PROGRAM Programa
VAR
    ToffPulse_1s : TON;
    TonPulse_1s : TON;
    ToffPulse_100ms : TON;
    TonPulse_100ms : TON;
    ToffPulse_2s : TON;
    TonPulse_2s : TON;
    ToffPulse_5s : TON;
    TonPulse_5s : TON;
    ToffPulse_10ms : TON;
    TonPulse_10ms : TON;
    ToffPulse_30s : TON;
    TonPulse_30s : TON;
    DelayRobotStep1 : TON;
    DelayRobotStep2 : TON;
    DelayRobotStep3 : TON;
    DelayRobotStep4 : TON;
    DelayRobotStep5 : TON;
    DelayRobotStep6 : TON;
    DelayRobotStep7 : TON;
    DelayRobotStep8 : TON;
    Motor110M1 : CmdLenzeI550;
    TimeResetAlarme : TON;
    Motor111M1 : CmdLenzeI550;
    Motor120M1 : CmdLenzeI550;
    Motor211M1 : CmdLenzeI550;
    Motor212M1 : CmdLenzeI550;
    Motor213M1 : CmdLenzeI550;
    Motor221M1 : CmdLenzeI550;
    Motor222M1 : CmdLenzeI550;
    Motor223M1 : CmdLenzeI550;
    Motor230M1 : CmdLenzeI550;
    Motor240M1 : CmdLenzeI550;
    Motor250M1 : CmdLenzeI550;
    Valve110V : CmdValve;
    Delay110M1Full : TON;
    Delay110VStep1 : TON;
    ncteste : BOOL;
    DelayAE110V : TON;
    Valve111V : CmdValve;
    DelayAE111V : TON;
    Delay111VStep4 : TON;
    DelayAE121V : TON;
    Valve121V : CmdValve;
    Delay121VStep4 : TON;
    DelayAE122V : TON;
    Delay122VStep4 : TON;
    DelayAE123V : TON;
    Valve122V : CmdValve;
    Delay123VStep4 : TON;
    DelayAE211V : TON;
    Valve211V : CmdValve;
    Delay211VStep1 : TON;
    DelayAE212V : TON;
    Valve212V : CmdValve;
    Delay212VStep1 : TON;
    DelayAE213V : TON;
    Valve213V : CmdValve;
    Delay213VStep1 : TON;
    Delay211M1Full : TON;
    Delay212M1Full : TON;
    Delay213M1Full : TON;
    Delay221M1Step2 : TON;
    Alarme_G_221M1 : CheckAlarmeEquip;
    Delay221M1Step4 : TimerPulse;
    Delay221M1Step9 : TON;
    Delay221M1Step11 : TimerPulse;
    Delay221M1Step16 : TimerPulse;
    Delay211M1Empty : TON;
    Delay212M1Empty : TON;
    Delay213M1Empty : TON;
    Delay211M1TimeOut : TON;
    Delay212M1TimeOut : TON;
    Delay213M1TimeOut : TON;
    Delay110M1TimeOut : TON;
    Alarme_G_230M1 : CheckAlarmeEquip;
    Delay230M1Step4 : TimerPulse;
    Delay230M1Step2 : TON;
    Delay221M1Step18 : TON;
    Delay230M1Step13 : TON;
    Delay230M1Step16 : TON;
    Delay221M1Step19 : TON;
    Alarme_G_222M1 : CheckAlarmeEquip;
    Delay222M1Step19 : TON;
    Delay222M1Step18 : TON;
    Delay222M1Step16 : TimerPulse;
    Delay222M1Step11 : TimerPulse;
    Delay222M1Step9 : TON;
    Delay222M1Step4 : TimerPulse;
    Delay222M1Step2 : TON;
    Alarme_G_223M1 : CheckAlarmeEquip;
    Delay223M1Step19 : TON;
    Delay223M1Step18 : TON;
    Delay223M1Step16 : TimerPulse;
    Delay223M1Step11 : TimerPulse;
    Delay223M1Step9 : TON;
    Delay223M1Step4 : TimerPulse;
    Delay223M1Step2 : TON;
    Delay111M1Step2 : TON;
    Delay111M1Step3 : TimerPulse;
    Delay111M1Step10 : TimerPulse;
    Delay111M1Step11 : TimerPulse;
    Delay111M1Step12 : TON;
    Delay111M1Step13 : TON;
    Delay111M1Step19 : TON;
    Delay111M1Step20 : TON;
    Read111U1 : EAN13Read;
    TimeOut111M1Step15 : TON;
    Delay111M1Step14 : TON;
    Delay120M1Step2 : TON;
    Delay120M1Step3 : TimerPulse;
    Delay120M1Step4 : TON;
    Delay120M1Step9 : TON;
    Delay120M1Step19 : TON;
    Delay111M1Step21 : TON;
    Delay120M1Step10 : TimerPulse;
    Delay120M1Step11 : TimerPulse;
    Delay120M1Step13 : TimerPulse;
    Delay120M1Step14 : TimerPulse;
    Delay120M1Step17 : TimerPulse;
    Delay120M1Step16 : TimerPulse;
    Alarme_G_240M1 : CheckAlarmeEquip;
    Delay240M1Step2 : TON;
    Delay240M1Step4 : TimerPulse;
    Delay240M1Step5 : TON;
    Delay240M1Step8 : TON;
    Delay240M1Step12 : TON;
    Alarme_G_250M1 : CheckAlarmeEquip;
    Delay250M1Step5 : TON;
    Delay250M1Step4 : TimerPulse;
    Delay250M1Step2 : TON;
    Delay250M1Step21 : TON;
    Delay250M1Step20 : TON;
    Delay250M1Step19 : TON;
    TimeOut250M1Step15 : TON;
    Delay250M1Step14 : TON;
    Delay250M1Step13 : TON;
    Delay250M1Step12 : TON;
    Delay250M1Step11 : TimerPulse;
    Delay250M1Step10 : TimerPulse;
    DelayAE251V : TON;
    Valve251V : CmdValve;
    Delay251VStep4 : TON;
    DelayAE252V : TON;
    Valve252V : CmdValve;
    Delay252VStep4 : TON;
    Delay250M1Step23 : TON;
    TimeMax251VStep3 : TON;
    TimeMax252VStep3 : TON;
    Delay250M1Step28 : TON;
    RstEthercat : ResetECError;
    RstPLC : ResetPLCError;
    CmdICM_540 : CmdICM;
    Motor540M1 : CmdMotor;
    Motor540M2 : CmdMotor;
    Motor610M1 : CmdMotor;
    Motor620M1 : CmdMotor;
    SystemTime : DATE_AND_TIME;  (* System Time on Gregorian date format *)
    year : INT;
    month : INT;
    day : INT;
    JD_aux01 : LINT;
    JD_aux02 : LINT;
    MCControllerErrorExists : BOOL;
    MCError_Level : UINT;
    MCError_Code : DWORD;
    ResetMCError_Servo : ResetMCError;
    MCR88_Power : MC_Power;
    MCR88_Power_Busy : BOOL;
    Motor310M1 : CmdMotor;
    Alarme_G_310M1 : CheckAlarmeEquip;
    Delay310M1Step2 : TON;
    Delay310M1Step4 : TimerPulse;
    Delay310M1Step5 : TON;
    Valve321V : CmdValve;
    FastStop320M1 : MC_Stop;
    Home320M1 : MC_Home;
    Move320M1ToPos0 : MC_MoveAbsolute;
    Move320M1ToPos1 : MC_MoveAbsolute;
    Move320M1ToPos2 : MC_MoveAbsolute;
    DelayGoToPos0 : TON;
    DelayGoToPos1 : TON;
    DelayGoToPos2 : TON;
    Delay310M1Step9 : TON;
    Delay310M1Step10 : TON;
    Delay310M1Step11 : TON;
    Delay310M1Step12 : TON;
    Delay310M1Step13 : TON;
    Delay310M1Step14 : TON;
    Delay310M1Step15 : TON;
    TempoIndexaçãoStep16 : TON;
    Delay310M1Step17 : TON;
    Delay310M1Step22 : TON;
    Read250U1 : EAN13Read;
    Check111U1 : CheckBarCode;
    Delay111U1Stp4 : TON;
    TempJulianDateES2 : LINT;
    DelayResetErro111U1 : TON;
    TimeOutRead111U1 : TON;
    DelayResetErro250U1 : TON;
    TimeOutRead250U1 : TON;
    Check250U1 : CheckBarCode;
    DelayAE321V : TON;
    DelayAuto310off : TOF;
    PedeDescargaToRobot : BOOL;  (* Existe um pedido de descarga para o Robot *)
    Delay221M1Step22 : TimerPulse;
    PedeDescargaToReject : BOOL;  (* Existe um pedido de descarga para os Rejeitados *)
    RdyToSendToRobot : BOOL;  (* Pronto a Enviar para Robot *)
    Delay221M1Step25 : TON;
    Delay221M1Step24 : TON;
    Delay222M1Step25 : TON;
    Delay222M1Step24 : TON;
    Delay222M1Step22 : TimerPulse;
    Delay223M1Step24 : TON;
    Delay223M1Step25 : TON;
    Delay223M1Step22 : TimerPulse;
    Delay231YS1 : TON;
    Delay223M1Step6 : TON;
    Delay250U1Stp3 : TON;
    Delay222M1Step6 : TON;
    Delay221M1Step6 : TON;
    TimeOut111M1Step9 : TON;
    Jog320M1 : MC_MoveJog;
    DZ_HMI_00 : TON;
    DZ_HMI_01 : TON;
    DZ_510M1_01 : TON;
    DZ_510M1_02 : TON;
    DZ_510M1_03 : TON;
    DZ_510M1_04 : TON;
    Motor510M1 : CmdMotor;
    DZ_510M1_06 : TON;
    DZ_510M1_07 : TON;
    If_520YS1 : BOOL;
    DZ_520M1_01 : TON;
    DZ_520M1_04 : TON;
    DZ_520M1_05 : TON;
    DZ_520M1_06 : TON;
    DZ_520M1_07 : TON;
    DZ_520M1_08 : TON;
    DZ_520M1_09 : TON;
    Motor520M1 : CmdMotor;
    Motor520M2 : CmdMotor;
    DZ_530M1_01 : TON;
    DZ_530M1_09 : TON;
    DZ_530M1_08 : TON;
    DZ_530M1_02 : TON;
    DZ_530M1_05 : TON;
    DZ_530M1_03 : TON;
    DZ_530M1_04 : TON;
    NumCodigosBarrasLidos : UINT;
    DZ_530M1_06 : TON;
    DZ_530M1_07 : TON;
    ReadString : string[128];
    DZ_530M1_10 : TON;
    Read530U1 : EAN13Read;
    Read530U2 : EAN13Read;
    DZ_540M1_01 : TON;
    DZ_540M1_02 : TON;
    DZ_540M1_03 : TON;
    DZ_540M1_04 : TON;
    DZ_540M1_05 : TON;
    DZ_550U1_01 : TON;
    DZ_550U1_02 : TON;
    DZ_550U1_03 : TON;
    DZ_550U1_04 : TON;
    DZ_550U1_05 : TON;
    DZ_550U1_06 : TON;
    DZ_550U1_07 : TON;
    DZ_550U1_08 : TON;
    DZ_550U1_09 : TON;
    DZ_550U1_11 : TON;
    DZ_550U1_10 : TON;
    DZ_610M1_01 : TON;
    DZ_610M1_02 : TON;
    DZ_610M1_03 : TON;
    DZ_610M1_04 : TON;
    DZ_610M1_05 : TON;
    DZ_620M1_01 : TON;
    DZ_620M1_02 : TON;
    DZ_620M1_03 : TON;
    DZ_620M1_04 : TON;
    DZ_620M1_05 : TON;
    DZ_630M1_01 : TON;
    DZ_630M1_02 : TON;
    DZ_630M1_03 : TON;
    Motor630M1 : CmdMotor;
    DZ_630M1_04 : TON;
    DZ_630M1_05 : TON;
    DZ_640M1_01 : TON;
    DZ_640M1_02 : TON;
    DZ_640M1_03 : TON;
    DZ_640M1_04 : TON;
    DZ_640M1_05 : TON;
    DZ_640M1_06 : TON;
    DZ_640M1_07 : TON;
    Motor640M1 : CmdMotor;
    Motor641M1 : CmdMotor;
    DZ_640M1_10 : TON;
    DZ_640M1_11 : TON;
    Motor640M2 : CmdMotor;
    DZ_640M2_01 : TON;
    DZ_640M2_02 : TON;
    DZ_640M2_03 : TON;
    DZ_640M2_04 : TON;
    DZ_640M2_05 : TON;
    DZ_640M2_06 : TON;
    DZ_640M2_07 : TON;
    Motor642M1 : CmdMotor;
    Motor643M1 : CmdMotor;
    DZ_640M2_08 : TON;
    DZ_640M2_09 : TON;
    DZ_640M2_11 : TON;
    DZ_640M2_12 : TON;
    FromG9SP_00 : WORD;
    DZ_020A1_01 : TON;
    DZ_020A1_02 : TON;
    FromG9SP_10 : WORD;
    CmdICM_520 : CmdICM;
    CmdICM_641 : CmdICM;
    CmdICM_643 : CmdICM;
    DZ_550U1_12 : TON;
    DZ_550U1_13 : TP;
    DZ_550U1_14 : TP;
    RebobinaAposNotOk : BOOL;
END_VAR
VAR_EXTERNAL
    Pulse_1s : BOOL;
    Pulse_100ms : BOOL;
    Pulse_2s : BOOL;
    Pulse_5s : BOOL;
    Pulse_10ms : BOOL;
    Pulse_30s : BOOL;
    StartRobot : BOOL;
    G_Robot : Grafcet;
    IFQ_330_DrivesOff : BOOL;
    IFQ_330_ConfMess : BOOL;
    IFQ_330_DrivesOn : BOOL;
    IFQ_330_ExtStart : BOOL;
    IFQ_330_MoveEnable : BOOL;
    IFQ_330_WORD1 : ARRAY[0..15] OF BOOL;
    IFQ_330_WatchDog : BOOL;
    IFI_330_WatchDog : BOOL;
    IFI_330_WORD1 : ARRAY[0..15] OF BOOL;
    IFI_330_In250 : BOOL;
    IFI_330_In310 : BOOL;
    IFQ_330_RdytoPick : BOOL;
    IFQ_330_RdytoPlace : BOOL;
    IFQ_330_Rst310 : BOOL;
    IFQ_330_NewData : BOOL;
    IFQ_330_DataOK : BOOL;
    IFQ_330_NotaType : WORD;
    IFI_330_NotaType : WORD;
    E009_TPDO4_mapping_parameter_CiA_Statusword_6041_00 : UINT;
    E009_RPDO4_mapping_parameter_Target_velocity_6042_00 : INT;
    E009_RPDO4_mapping_parameter_CiA_Controlword_6040_00 : UINT;
    E003_TPDO4_mapping_parameter_CiA_Statusword_6041_00 : UINT;
    E003_RPDO4_mapping_parameter_Target_velocity_6042_00 : INT;
    E003_RPDO4_mapping_parameter_CiA_Controlword_6040_00 : UINT;
    E003_RPDO6_mapping_parameter_CiA_Acceleration_ms_2917_00 : UINT;
    E003_RPDO6_mapping_parameter_CiA_Deceleration_ms_2918_00 : UINT;
    E002_TPDO4_mapping_parameter_CiA_Statusword_6041_00 : UINT;
    E002_RPDO4_mapping_parameter_Target_velocity_6042_00 : INT;
    E002_RPDO6_mapping_parameter_CiA_Acceleration_ms_2917_00 : UINT;
    E002_RPDO6_mapping_parameter_CiA_Deceleration_ms_2918_00 : UINT;
    E002_RPDO4_mapping_parameter_CiA_Controlword_6040_00 : UINT;
    A_110M1 : AlarmeGeralEquipamento;
    E_110M1 : Event;
    D_110M1 : DataMotor;
    IFQ_330_StopRequest : BOOL;
    IFI_330_InHome : BOOL;
    IFI_330_RstDone : BOOL;
    IFI_330_StopRequestDone : BOOL;
    IFI_330_ProductLost : BOOL;
    IFI_330_GeneralError : BOOL;
    IFI_330_BoxComplete : BOOL;
    IFI_330_OpenTool : BOOL;
    IFI_330_CloseTool : BOOL;
    IFQ_330_330YS1 : BOOL;
    IFQ_330_330YS2 : BOOL;
    IFQ_330_330XS1 : BOOL;
    IFQ_330_RstProdLost : BOOL;
    ResetAlarmes : BOOL;
    T_Reset : BOOL;
    D_111M1 : DataMotor;
    A_111M1 : AlarmeGeralEquipamento;
    E_111M1 : Event;
    D_120M1 : DataMotor;
    A_120M1 : AlarmeGeralEquipamento;
    E_120M1 : Event;
    E004_TPDO4_mapping_parameter_CiA_Statusword_6041_00 : UINT;
    E004_RPDO4_mapping_parameter_Target_velocity_6042_00 : INT;
    E004_RPDO6_mapping_parameter_CiA_Acceleration_ms_2917_00 : UINT;
    E004_RPDO6_mapping_parameter_CiA_Deceleration_ms_2918_00 : UINT;
    E004_RPDO4_mapping_parameter_CiA_Controlword_6040_00 : UINT;
    D_211M1 : DataMotor;
    A_211M1 : AlarmeGeralEquipamento;
    E_211M1 : Event;
    E005_TPDO4_mapping_parameter_CiA_Statusword_6041_00 : UINT;
    E005_RPDO4_mapping_parameter_Target_velocity_6042_00 : INT;
    E005_RPDO6_mapping_parameter_CiA_Acceleration_ms_2917_00 : UINT;
    E005_RPDO6_mapping_parameter_CiA_Deceleration_ms_2918_00 : UINT;
    E005_RPDO4_mapping_parameter_CiA_Controlword_6040_00 : UINT;
    D_212M1 : DataMotor;
    A_212M1 : AlarmeGeralEquipamento;
    E_212M1 : Event;
    E006_TPDO4_mapping_parameter_CiA_Statusword_6041_00 : UINT;
    E006_RPDO4_mapping_parameter_Target_velocity_6042_00 : INT;
    E006_RPDO6_mapping_parameter_CiA_Acceleration_ms_2917_00 : UINT;
    E006_RPDO6_mapping_parameter_CiA_Deceleration_ms_2918_00 : UINT;
    E006_RPDO4_mapping_parameter_CiA_Controlword_6040_00 : UINT;
    D_213M1 : DataMotor;
    A_213M1 : AlarmeGeralEquipamento;
    E_213M1 : Event;
    E007_TPDO4_mapping_parameter_CiA_Statusword_6041_00 : UINT;
    E007_RPDO4_mapping_parameter_Target_velocity_6042_00 : INT;
    E007_RPDO6_mapping_parameter_CiA_Acceleration_ms_2917_00 : UINT;
    E007_RPDO6_mapping_parameter_CiA_Deceleration_ms_2918_00 : UINT;
    E007_RPDO4_mapping_parameter_CiA_Controlword_6040_00 : UINT;
    D_221M1 : DataMotor;
    A_221M1 : AlarmeGeralEquipamento;
    E_221M1 : Event;
    E008_TPDO4_mapping_parameter_CiA_Statusword_6041_00 : UINT;
    E008_RPDO4_mapping_parameter_Target_velocity_6042_00 : INT;
    E008_RPDO6_mapping_parameter_CiA_Acceleration_ms_2917_00 : UINT;
    E008_RPDO6_mapping_parameter_CiA_Deceleration_ms_2918_00 : UINT;
    E008_RPDO4_mapping_parameter_CiA_Controlword_6040_00 : UINT;
    D_222M1 : DataMotor;
    A_222M1 : AlarmeGeralEquipamento;
    E009_RPDO6_mapping_parameter_CiA_Acceleration_ms_2917_00 : UINT;
    E009_RPDO6_mapping_parameter_CiA_Deceleration_ms_2918_00 : UINT;
    D_223M1 : DataMotor;
    A_223M1 : AlarmeGeralEquipamento;
    E_223M1 : Event;
    E010_TPDO4_mapping_parameter_CiA_Statusword_6041_00 : UINT;
    E010_RPDO4_mapping_parameter_Target_velocity_6042_00 : INT;
    E010_RPDO6_mapping_parameter_CiA_Acceleration_ms_2917_00 : UINT;
    E010_RPDO6_mapping_parameter_CiA_Deceleration_ms_2918_00 : UINT;
    E010_RPDO4_mapping_parameter_CiA_Controlword_6040_00 : UINT;
    E_222M1 : Event;
    D_230M1 : DataMotor;
    A_230M1 : AlarmeGeralEquipamento;
    E_230M1 : Event;
    E011_TPDO4_mapping_parameter_CiA_Statusword_6041_00 : UINT;
    E011_RPDO4_mapping_parameter_Target_velocity_6042_00 : INT;
    E011_RPDO6_mapping_parameter_CiA_Acceleration_ms_2917_00 : UINT;
    E011_RPDO6_mapping_parameter_CiA_Deceleration_ms_2918_00 : UINT;
    E011_RPDO4_mapping_parameter_CiA_Controlword_6040_00 : UINT;
    D_240M1 : DataMotor;
    A_240M1 : AlarmeGeralEquipamento;
    E_240M1 : Event;
    E012_TPDO4_mapping_parameter_CiA_Statusword_6041_00 : UINT;
    E012_RPDO4_mapping_parameter_Target_velocity_6042_00 : INT;
    E012_RPDO6_mapping_parameter_CiA_Acceleration_ms_2917_00 : UINT;
    E012_RPDO6_mapping_parameter_CiA_Deceleration_ms_2918_00 : UINT;
    E012_RPDO4_mapping_parameter_CiA_Controlword_6040_00 : UINT;
    D_250M1 : DataMotor;
    A_250M1 : AlarmeGeralEquipamento;
    E_250M1 : Event;
    E013_TPDO4_mapping_parameter_CiA_Statusword_6041_00 : UINT;
    E013_RPDO4_mapping_parameter_Target_velocity_6042_00 : INT;
    E013_RPDO6_mapping_parameter_CiA_Acceleration_ms_2917_00 : UINT;
    E013_RPDO6_mapping_parameter_CiA_Deceleration_ms_2918_00 : UINT;
    E013_RPDO4_mapping_parameter_CiA_Controlword_6040_00 : UINT;
    D_110V : DataValve;
    A_110V : AlarmeGeralEquipamento;
    E_110V : Event;
    MachineAuto : BOOL;
    Zona110Auto : BOOL;
    Zona120Auto : BOOL;
    MachineOn : BOOL;
    DT_110M1 : DataTransport;
    I_110YS1 : BOOL;
    I_110YS2 : BOOL;
    I_110XS1 : BOOL;
    G_110V : GrafcetBatente;
    I_110XS2 : BOOL;
    CondGeraisOK : BOOL;
    Exec_G_110V : BOOL;
    Q_110V1 : BOOL;
    Q_110V2 : BOOL;
    Q_900V1 : BOOL;
    D_111V : DataValve;
    Exec_G_111V : BOOL;
    G_111V : GrafcetEmpurrador;
    A_111V : AlarmeGeralEquipamento;
    E_111V : Event;
    Q_111V1 : BOOL;
    Q_111V2 : BOOL;
    I_111XS1 : BOOL;
    I_111XS2 : BOOL;
    D_121V : DataValve;
    I_121XS1 : BOOL;
    I_121XS2 : BOOL;
    Q_121V1 : BOOL;
    Q_121V2 : BOOL;
    A_121V : AlarmeGeralEquipamento;
    E_121V : Event;
    Exec_G_121V : BOOL;
    G_121V : GrafcetEmpurrador;
    D_122V : DataValve;
    I_122XS1 : BOOL;
    I_122XS2 : BOOL;
    A_122V : AlarmeGeralEquipamento;
    Exec_G_122V : BOOL;
    G_122V : GrafcetEmpurrador;
    E_122V : Event;
    Q_122V1 : BOOL;
    Q_122V2 : BOOL;
    D_123V : DataValve;
    I_123XS1 : BOOL;
    I_123XS2 : BOOL;
    A_123V : AlarmeGeralEquipamento;
    Q_123V1 : BOOL;
    Q_123V2 : BOOL;
    E_123V : Event;
    Exec_G_123V : BOOL;
    G_123V : GrafcetEmpurrador;
    ZonaBuffer1Auto : BOOL;
    D_211V : DataValve;
    I_211XS1 : BOOL;
    I_211XS2 : BOOL;
    A_211V : AlarmeGeralEquipamento;
    Q_211V1 : BOOL;
    Q_211V2 : BOOL;
    E_211V : Event;
    Exec_G_211V : BOOL;
    G_211V : GrafcetBatente;
    I_211YS2 : BOOL;
    ZonaBuffer2Auto : BOOL;
    D_212V : DataValve;
    I_212XS1 : BOOL;
    I_212XS2 : BOOL;
    A_212V : AlarmeGeralEquipamento;
    Q_212V1 : BOOL;
    Q_212V2 : BOOL;
    E_212V : Event;
    G_212V : GrafcetBatente;
    Exec_G_212V : BOOL;
    I_212YS2 : BOOL;
    ZonaBuffer3Auto : BOOL;
    D_213V : DataValve;
    I_213XS1 : BOOL;
    I_213XS2 : BOOL;
    A_213V : AlarmeGeralEquipamento;
    Q_213V2 : BOOL;
    Q_213V1 : BOOL;
    E_213V : Event;
    Exec_G_213V : BOOL;
    G_213V : GrafcetBatente;
    I_213YS2 : BOOL;
    DT_211M1 : DataTransport;
    I_211YS1 : BOOL;
    DT_212M1 : DataTransport;
    I_212YS1 : BOOL;
    DT_213M1 : DataTransport;
    I_213YS1 : BOOL;
    Exec_G_221M1 : BOOL;
    G_221M1 : GrafcetAcumula;
    I_221YS2 : BOOL;
    AG_221M1 : Alarme;
    DP_221M1 : DataProd;
    DP_211M1 : DataProd;
    DP_212M1 : DataProd;
    DP_213M1 : DataProd;
    I_330YS1 : BOOL;
    I_330YS2 : BOOL;
    I_330XS1 : BOOL;
    Q_330V1 : BOOL;
    Q_330V2 : BOOL;
    I_251YS1 : BOOL;
    I_251XS1 : BOOL;
    G_222M1 : GrafcetAcumula;
    G_223M1 : GrafcetAcumula;
    Zona230Auto : BOOL;
    AG_230M1 : Alarme;
    Exec_G_230M1 : BOOL;
    G_230M1 : Grafcet230M1;
    I_230YS2 : BOOL;
    DP_230M1 : DataProd;
    I_231YS1 : BOOL;
    AG_222M1 : Alarme;
    I_222YS2 : BOOL;
    Exec_G_222M1 : BOOL;
    DP_222M1 : DataProd;
    AG_223M1 : Alarme;
    I_223YS3 : BOOL;
    Exec_G_223M1 : BOOL;
    DP_223M1 : DataProd;
    Zona240Auto : BOOL;
    Zona250Auto : BOOL;
    Exec_G_111M1 : BOOL;
    G_111M1 : Grafcet111M1;
    I_111YS1 : BOOL;
    I_111YS2 : BOOL;
    DP_111M1 : DataProd;
    Q_111U1TRG : BOOL;
    I_IFM01_BarCodeReader_111U1 : ARRAY[0..449] OF BYTE;
    Exec_G_120M1 : BOOL;
    G_120M1 : Grafcet120M1;
    I_124YS1 : BOOL;
    I_121YS1 : BOOL;
    I_122YS1 : BOOL;
    I_123YS1 : BOOL;
    DP_120M1 : DataProd;
    I_111U1OK : BOOL;
    Exec_G_240M1 : BOOL;
    G_240M1 : Grafcet240M1;
    DP_240M1 : DataProd;
    AG_240M1 : Alarme;
    I_240YS2 : BOOL;
    G_250M1 : Grafcet250M1;
    AG_250M1 : Alarme;
    Exec_G_250M1 : BOOL;
    I_250YS2 : BOOL;
    DP_250M1 : DataProd;
    I_251XS2 : BOOL;
    I_250YS1 : BOOL;
    D_251V : DataValve;
    A_251V : AlarmeGeralEquipamento;
    Q_251V1 : BOOL;
    Q_251V2 : BOOL;
    E_251V : Event;
    Exec_G_251V : BOOL;
    G_251V : GrafcetEmpurrador;
    I_252XS2 : BOOL;
    D_252V : DataValve;
    I_252XS1 : BOOL;
    Q_252V1 : BOOL;
    Q_252V2 : BOOL;
    A_252V : AlarmeGeralEquipamento;
    E_252V : Event;
    Exec_G_252V : BOOL;
    G_252V : GrafcetEmpurrador;
    A_Geral : AlarmeGeralLinha;
    I_900PS1 : BOOL;
    HMI_EtiquetaMilheiro_01 : STRING[256];
    HMI_EtiquetaMilheiro_02 : STRING[256];
    HMI_EtiquetaMilheiro_03 : STRING[256];
    HMI_EtiquetaMilheiro_04 : STRING[256];
    HMI_EtiquetaMilheiro_05 : STRING[256];
    HMI_EtiquetaMilheiro_06 : STRING[256];
    HMI_EtiquetaMilheiro_07 : STRING[256];
    HMI_EtiquetaMilheiro_08 : STRING[256];
    HMI_EtiquetaMilheiro_09 : STRING[256];
    HMI_EtiquetaMilheiro_10 : STRING[256];
    HMI_PleaseCreateBox : BOOL;
    HMI_PleasePrintBoxId : BOOL;
    HMI_CreateBoxOK : BOOL;
    HMI_CreateBoxNOK : BOOL;
    HMI_PrintOK : BOOL;
    HMI_PrintNOK : BOOL;
    HMI_Maquina : string[256];
    I_320XS1 : BOOL;
    Q_320XS1 : BOOL;
    I_320XS2 : BOOL;
    I_320XS3 : BOOL;
    Q_320XS2 : BOOL;
    Q_320XS3 : BOOL;
    Q_321V1 : BOOL;
    I_Interroll_540 : In_EIPMulticontrol;
    Q_Interroll_540 : Out_EIPMulticontrol;
    I_540YS1 : BOOL;
    I_540YS2 : BOOL;
    D_540M1 : DataMotor;
    A_540M1 : AlarmeGeralEquipamento;
    E_540M1 : Event;
    D_540M2 : DataMotor;
    A_540M2 : AlarmeGeralEquipamento;
    E_540M2 : Event;
    D_610M1 : DataMotor;
    A_610M1 : AlarmeGeralEquipamento;
    E_610M1 : Event;
    D_620M1 : DataMotor;
    A_620M1 : AlarmeGeralEquipamento;
    E_620M1 : Event;
    I_540XS1 : BOOL;
    I_540XS2 : BOOL;
    A_320M1 : AlarmeGeralEquipamento;
END_VAR
VAR_EXTERNAL CONSTANT
    MC_Axis320M1 : _sAXIS_REF;
END_VAR
VAR_EXTERNAL
    E015_Error_code : WORD;
    JulianDate : LINT;
    Q_321V2 : BOOL;
    Zona310Auto : BOOL;
    D_310M1 : DataMotor;
    Exec_G_310M1 : BOOL;
    G_310M1 : Grafcet310M1;
    A_310M1 : AlarmeGeralEquipamento;
    E_310M1 : Event;
    AG_310M1 : Alarme;
    Q_310VL1 : BOOL;
    Q_310VL2 : BOOL;
    I_321XS2 : BOOL;
    I_321XS1 : BOOL;
    I_310YS2 : BOOL;
    D_321V : DataValve;
    A_321V : AlarmeGeralEquipamento;
    E_321V : Event;
    D_320M1 : DataServo;
    DP_320M1 : Position;
    WidthMax320M1 : LREAL;
    Width5Euro : LREAL;
    Width10Euro : LREAL;
    Width20Euro : LREAL;
    Width50Euro : LREAL;
    Width100Euro : LREAL;
    Width200Euro : LREAL;
    Width500Euro : LREAL;
    DP_310M1 : DataProd;
    I_400Auto : BOOL;
    DataRead111U1 : DataLCB;
    DataRead250U1 : DataLCB;
    I_IFM01_BarCodeReader_250U1 : ARRAY[0..449] OF BYTE;
    I_250U1OK : BOOL;
    Q_250U1TRG : BOOL;
    Code111U1OK : BOOL;
    Code111U1NOK : BOOL;
    Code250U1OK : BOOL;
    Code250U1NOK : BOOL;
    Exec_G_111U1 : BOOL;
    G_111U1 : Grafcet111U1;
    TRG_111U1 : BOOL;
    A_111U1 : Alarme;
    Erro_111U1 : BOOL;
    JulianDateES1 : UINT;
    JulianDateES2 : UINT;
    ds : _sDT;  (* DateStruct of the Var SystemTime to use on "Julian Date" *)
    TRG_250U1 : BOOL;
    Erro_250U1 : BOOL;
    Exec_G_250U1 : BOOL;
    G_250U1 : Grafcet250U1;
    A_250U1 : Alarme;
    D_Buffer1 : DataBuffer;
    D_Buffer2 : DataBuffer;
    D_Buffer3 : DataBuffer;
    Q_900LG : BOOL;
    Q_900LR : BOOL;
    I_300HS1 : BOOL;
    I_300HS2 : BOOL;
    Zona300On : BOOL;
    CondGerais300OK : BOOL;
    WatchDogHMI : BOOL;
    ErroComunicacaoPC : BOOL;
    D_510M1 : DataMotor;
    Exec_G_510M1 : BOOL;
    G_510M1 : Grafcet510M1;
    I_510YS2 : BOOL;
    I_510YS1 : BOOL;
    A_510M1 : AlarmeGeralEquipamento;
    G_520M1 : Grafcet520M1;
    D_520M1 : DataMotor;
    Exec_G_520M1 : BOOL;
    E_510M1 : Event;
    I_520XS1 : BOOL;
    I_520XS2 : BOOL;
    Zona510520Auto : BOOL;
    D_520M2 : DataMotor;
    I_520YS1 : BOOL;
    A_520M1 : AlarmeGeralEquipamento;
    Q_520V1 : BOOL;
    Q_520V2 : BOOL;
    G_530M1 : Grafcet530M1;
    D_530M1 : DataMotor;
    E_520M1 : Event;
    A_520M2 : AlarmeGeralEquipamento;
    E_520M2 : Event;
    Exec_G_530M1 : BOOL;
    A_530M1 : AlarmeGeralEquipamento;
    I_530YS3 : BOOL;
    G_550U1 : Grafcet550U1;
    Exec_G_550U1 : BOOL;
    I_530YS1 : BOOL;
    I_530YS2 : BOOL;
    Q_530VL1 : BOOL;
    Q_530VL2 : BOOL;
    DataRead530U1 : DataLCB;
    TRG_530U1 : BOOL;
    TRG_530U2 : BOOL;
    DataRead530U2 : DataLCB;
    G_540M1 : Grafcet540M1;
    Zona530Auto : BOOL;
    J02_EstbTargetSta : ARRAY[0..63] OF BOOL;
    Q_530U1TRG : BOOL;
    I_IFM01_BarCodeReader_530U1 : ARRAY[0..449] OF BYTE;
    I_530U1OK : BOOL;
    Q_530U2TRG : BOOL;
    I_IFM01_BarCodeReader_530U2 : ARRAY[0..449] OF BYTE;
    I_530U2OK : BOOL;
    Exec_G_540M1 : BOOL;
    Q_540V1 : BOOL;
    Q_540V2 : BOOL;
    G_610M1 : Grafcet6X0M1_Transport;
    Zona540Auto : BOOL;
    A_550U : AlarmeGeralEquipamento;
    I_550Error : BOOL;
    I_553XS2 : BOOL;
    I_550Feed : BOOL;
    Q_553V2 : BOOL;
    Q_553V1 : BOOL;
    Q_551V1 : BOOL;
    Q_552V1 : BOOL;
    Q_550M1 : BOOL;
    Zona550Auto : BOOL;
    I_550YS1 : BOOL;
    Q_550LG : BOOL;
    Q_550LR : BOOL;
    I_550PS1 : BOOL;
    I_610YS2 : BOOL;
    Zona600Auto : BOOL;
    Exec_G_610M1 : BOOL;
    G_620M1 : Grafcet6X0M1_Transport;
    I_620YS2 : BOOL;
    Exec_G_620M1 : BOOL;
    G_630M1 : Grafcet6X0M1_Transport;
    Exec_G_630M1 : BOOL;
    D_630M1 : DataMotor;
    A_630M1 : AlarmeGeralEquipamento;
    E_630M1 : Event;
    G_640M1 : Grafcet6X0M1_Transport_Com2Transfer;
    I_630YS2 : BOOL;
    D_640M1 : DataMotor;
    D_641M1 : DataMotor;
    A_640M1 : AlarmeGeralEquipamento;
    A_641M1 : AlarmeGeralEquipamento;
    G_640M2 : Grafcet6X0M1_Transport_Com2Transfer;
    Exec_G_640M1 : BOOL;
    I_650YS1 : BOOL;
    E_640M1 : Event;
    Q_641V1 : BOOL;
    Q_641V2 : BOOL;
    E_641M1 : Event;
    I_641YS1 : BOOL;
    I_640YS2 : BOOL;
    I_641YS2 : BOOL;
    I_641XS1 : BOOL;
    I_641XS2 : BOOL;
    D_640M2 : DataMotor;
    D_642M1 : DataMotor;
    D_643M1 : DataMotor;
    A_640M2 : AlarmeGeralEquipamento;
    A_642M1 : AlarmeGeralEquipamento;
    A_643M1 : AlarmeGeralEquipamento;
    Exec_G_640M2 : BOOL;
    E_640M2 : Event;
    E_642M1 : Event;
    E_643M1 : Event;
    Q_642V1 : BOOL;
    Q_642V2 : BOOL;
    Q_643V1 : BOOL;
    Q_643V2 : BOOL;
    I_642YS1 : BOOL;
    I_642YS2 : BOOL;
    I_643YS2 : BOOL;
    I_643YS1 : BOOL;
    I_642XS2 : BOOL;
    I_642XS1 : BOOL;
    I_643XS2 : BOOL;
    I_643XS1 : BOOL;
    I_FromG9SP_100 : ARRAY[0..67] OF byte;
    SafetyIn : SafetyIn_struct;
    Q_ToG9SP_101 : ARRAY[0..5] OF byte;
    SafetyOut : SafetyOut_struct;
    A_020A1 : AlarmeGeralEquipamento;
    I_Interroll_520 : In_EIPMulticontrol;
    Q_Interroll_520 : Out_EIPMulticontrol;
    I_Interroll_641 : In_EIPMulticontrol;
    Q_Interroll_641 : Out_EIPMulticontrol;
    I_Interroll_643 : In_EIPMulticontrol;
    Q_Interroll_643 : Out_EIPMulticontrol;
    MachineID530M1 : UINT;
    MachineID540M1 : UINT;
    MachineID610M1 : UINT;
    MachineID620M1 : UINT;
    MachineID630M1 : UINT;
    MachineID640M1 : UINT;
    MachineID640M2 : UINT;
END_VAR
VAR
    _e1 : R_TRIG;
    _e2 : R_TRIG;
    _t3 : BOOL;
    _p4 : BOOL;
    _p5 : BOOL;
    _p6 : BOOL;
    _p7 : BOOL;
    _p8 : BOOL;
    _p9 : BOOL;
    _p10 : BOOL;
    _p11 : BOOL;
    _p12 : BOOL;
    _p13 : BOOL;
    _p14 : BOOL;
    _p15 : BOOL;
    _p16 : BOOL;
    _p17 : BOOL;
    _p18 : BOOL;
    _p19 : BOOL;
    _p20 : BOOL;
    _p21 : BOOL;
    _p22 : BOOL;
    _p23 : BOOL;
    _p24 : BOOL;
    _p25 : BOOL;
    _p26 : BOOL;
    _p27 : BOOL;
    _p28 : BOOL;
    _p29 : BOOL;
    _p30 : BOOL;
    _p31 : BOOL;
    _p32 : BOOL;
    _p33 : BOOL;
    _p34 : BOOL;
    _p35 : BOOL;
    _e36 : R_TRIG;
    _p37 : BOOL;
    _p38 : BOOL;
    _p39 : BOOL;
    _p40 : BOOL;
    _p41 : BOOL;
    _p42 : BOOL;
    _p43 : BOOL;
    _p44 : BOOL;
    _p45 : BOOL;
    _p46 : BOOL;
    _p47 : BOOL;
    _p48 : BOOL;
    _p49 : BOOL;
    _p50 : BOOL;
    _p51 : BOOL;
    _p52 : BOOL;
    _p53 : BOOL;
    _p54 : BOOL;
    _p55 : BOOL;
    _p56 : BOOL;
    _p57 : BOOL;
    _p58 : BOOL;
    _p59 : BOOL;
    _p60 : BOOL;
    _p61 : BOOL;
    _e62 : R_TRIG;
    _e63 : F_TRIG;
    _p64 : BOOL;
    _p65 : BOOL;
    _p66 : BOOL;
    _p67 : BOOL;
    _p68 : BOOL;
    _p69 : BOOL;
    _e70 : R_TRIG;
    _e71 : F_TRIG;
    _p72 : BOOL;
    _p73 : BOOL;
    _p74 : BOOL;
    _p75 : BOOL;
    _p76 : BOOL;
    _p77 : BOOL;
    _e78 : R_TRIG;
    _e79 : F_TRIG;
    _p80 : BOOL;
    _p81 : BOOL;
    _p82 : BOOL;
    _p83 : BOOL;
    _p84 : BOOL;
    _p85 : BOOL;
    _e86 : R_TRIG;
    _e87 : R_TRIG;
    _e88 : R_TRIG;
    _p89 : BOOL;
    _p90 : BOOL;
    _p91 : BOOL;
    _p92 : BOOL;
    _p93 : BOOL;
    _p94 : BOOL;
    _p95 : BOOL;
    _p96 : BOOL;
    _p97 : BOOL;
    _p98 : BOOL;
    _p99 : BOOL;
    _p100 : BOOL;
    _p101 : BOOL;
    _p102 : BOOL;
    _p103 : BOOL;
    _p104 : BOOL;
    _p105 : BOOL;
    _p106 : BOOL;
    _p107 : BOOL;
    _p108 : BOOL;
    _p109 : BOOL;
    _p110 : BOOL;
    _p111 : BOOL;
    _p112 : BOOL;
    _p113 : BOOL;
    _p114 : BOOL;
    _p115 : BOOL;
    _p116 : BOOL;
    _p117 : BOOL;
    _p118 : BOOL;
    _p119 : BOOL;
    _p120 : BOOL;
    _p121 : BOOL;
    _p122 : BOOL;
    _p123 : BOOL;
    _p124 : BOOL;
    _p125 : BOOL;
    _p126 : BOOL;
    _p127 : BOOL;
    _p128 : BOOL;
    _p129 : BOOL;
    _p130 : BOOL;
    _p131 : BOOL;
    _p132 : BOOL;
    _p133 : BOOL;
    _p134 : BOOL;
    _p135 : BOOL;
    _p136 : BOOL;
    _p137 : BOOL;
    _p138 : BOOL;
    _p139 : BOOL;
    _p140 : BOOL;
    _p141 : BOOL;
    _p142 : BOOL;
    _p143 : BOOL;
    _p144 : BOOL;
    _p145 : BOOL;
    _p146 : BOOL;
    _p147 : BOOL;
    _p148 : BOOL;
    _p149 : BOOL;
    _p150 : BOOL;
    _p151 : BOOL;
    _p152 : BOOL;
    _p153 : BOOL;
    _p154 : BOOL;
    _p155 : BOOL;
    _p156 : BOOL;
    _p157 : BOOL;
    _p158 : BOOL;
    _p159 : BOOL;
    _p160 : BOOL;
    _p161 : BOOL;
    _p162 : BOOL;
    _p163 : BOOL;
    _p164 : BOOL;
    _p165 : BOOL;
    _p166 : BOOL;
    _p167 : BOOL;
    _p168 : BOOL;
    _p169 : BOOL;
    _p170 : BOOL;
    _p171 : BOOL;
    _p172 : BOOL;
    _p173 : BOOL;
    _p174 : BOOL;
    _p175 : BOOL;
    _p176 : BOOL;
    _e177 : R_TRIG;
    _p178 : BOOL;
    _p179 : BOOL;
    _p180 : BOOL;
    _p181 : BOOL;
    _p182 : BOOL;
    _p183 : BOOL;
    _p184 : BOOL;
    _p185 : BOOL;
    _p186 : BOOL;
    _p187 : BOOL;
    _p188 : BOOL;
    _p189 : BOOL;
    _p190 : BOOL;
    _p191 : BOOL;
    _p192 : BOOL;
    _p193 : BOOL;
    _p194 : BOOL;
    _p195 : BOOL;
    _e196 : F_TRIG;
    _e197 : R_TRIG;
    _p198 : BOOL;
    _p199 : BOOL;
    _p200 : BOOL;
    _p201 : BOOL;
    _p202 : BOOL;
    _p203 : BOOL;
    _e204 : R_TRIG;
    _e205 : R_TRIG;
    _p206 : BOOL;
    _p207 : BOOL;
    _p208 : BOOL;
    _p209 : BOOL;
    _p210 : BOOL;
    _p211 : BOOL;
    _p212 : BOOL;
    _p213 : BOOL;
    _p214 : BOOL;
    _p215 : BOOL;
    _p216 : BOOL;
    _p217 : BOOL;
    _p218 : BOOL;
    _p219 : BOOL;
    _p220 : BOOL;
    _p221 : BOOL;
    _p222 : BOOL;
    _p223 : BOOL;
    _p224 : BOOL;
    _p225 : BOOL;
    _p226 : BOOL;
    _p227 : BOOL;
    _p228 : BOOL;
    _p229 : BOOL;
    _p230 : BOOL;
    _p231 : BOOL;
    _p232 : BOOL;
    _p233 : BOOL;
    _p234 : BOOL;
    _p235 : BOOL;
    _p236 : BOOL;
    _p237 : BOOL;
    _p238 : BOOL;
    _p239 : BOOL;
    _p240 : BOOL;
    _p241 : BOOL;
    _p242 : BOOL;
    _p243 : BOOL;
    _p244 : BOOL;
    _p245 : BOOL;
    _p246 : BOOL;
    _e247 : R_TRIG;
    _p248 : BOOL;
    _e249 : R_TRIG;
    _p250 : BOOL;
    _e251 : R_TRIG;
    _p252 : BOOL;
    _p253 : BOOL;
    _p254 : BOOL;
    _p255 : BOOL;
    _p256 : BOOL;
    _p257 : BOOL;
    _p258 : BOOL;
    _p259 : BOOL;
    _e260 : F_TRIG;
    _e261 : F_TRIG;
    _e262 : R_TRIG;
    _e263 : R_TRIG;
    _e264 : F_TRIG;
    _e265 : F_TRIG;
    _p266 : BOOL;
    _p267 : BOOL;
    _p268 : BOOL;
    _p269 : BOOL;
    _p270 : BOOL;
    _e271 : R_TRIG;
    _p272 : BOOL;
    _p273 : BOOL;
    _p274 : BOOL;
    _p275 : BOOL;
    _p276 : BOOL;
    _p277 : BOOL;
    _p278 : BOOL;
    _e279 : R_TRIG;
    _p280 : BOOL;
    _p281 : BOOL;
    _e282 : R_TRIG;
    _p283 : BOOL;
    _p284 : BOOL;
    _p285 : BOOL;
    _p286 : BOOL;
    _p287 : BOOL;
    _e288 : R_TRIG;
    _p289 : BOOL;
    _p290 : BOOL;
    _e291 : R_TRIG;
    _p292 : BOOL;
    _p293 : BOOL;
    _p294 : BOOL;
    _p295 : BOOL;
    _e296 : R_TRIG;
    _p297 : BOOL;
    _e298 : R_TRIG;
    _e299 : R_TRIG;
    _p300 : BOOL;
    _p301 : BOOL;
    _p302 : BOOL;
    _e303 : R_TRIG;
    _p304 : BOOL;
    _e305 : R_TRIG;
    _t306 : BOOL;
END_VAR

(* Section Pulses: ladder, written here as Structured Text *)

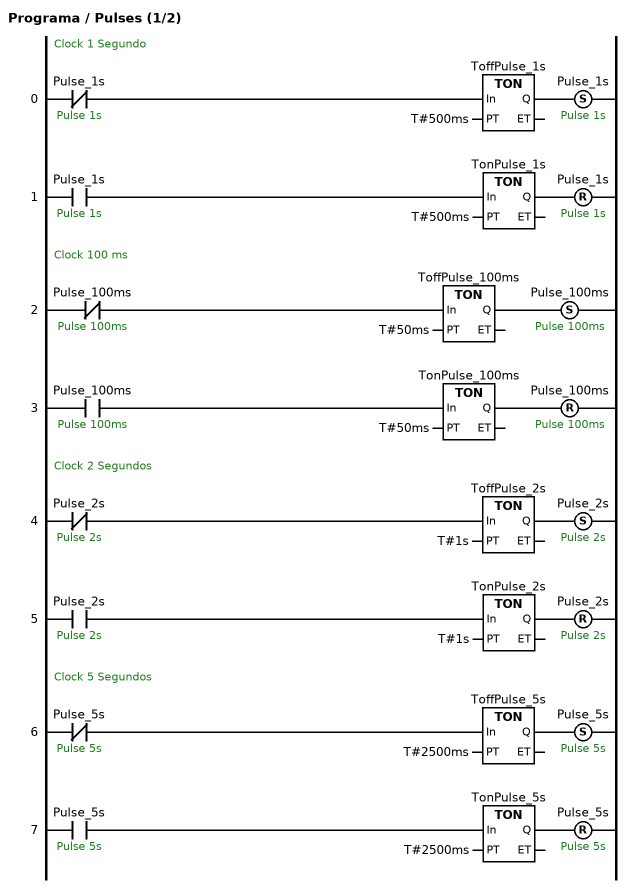
(* Rung 0: Clock 1 Segundo *)
ToffPulse_1s(In := NOT Pulse_1s, PT := T#500ms);
IF ToffPulse_1s.Q THEN Pulse_1s := TRUE; END_IF;
(* Rung 1 *)
TonPulse_1s(In := Pulse_1s, PT := T#500ms);
IF TonPulse_1s.Q THEN Pulse_1s := FALSE; END_IF;
(* Rung 2: Clock 100 ms *)
ToffPulse_100ms(In := NOT Pulse_100ms, PT := T#50ms);
IF ToffPulse_100ms.Q THEN Pulse_100ms := TRUE; END_IF;
(* Rung 3 *)
TonPulse_100ms(In := Pulse_100ms, PT := T#50ms);
IF TonPulse_100ms.Q THEN Pulse_100ms := FALSE; END_IF;
(* Rung 4: Clock 2 Segundos *)
ToffPulse_2s(In := NOT Pulse_2s, PT := T#1s);
IF ToffPulse_2s.Q THEN Pulse_2s := TRUE; END_IF;
(* Rung 5 *)
TonPulse_2s(In := Pulse_2s, PT := T#1s);
IF TonPulse_2s.Q THEN Pulse_2s := FALSE; END_IF;
(* Rung 6: Clock 5 Segundos *)
ToffPulse_5s(In := NOT Pulse_5s, PT := T#2500ms);
IF ToffPulse_5s.Q THEN Pulse_5s := TRUE; END_IF;
(* Rung 7 *)
TonPulse_5s(In := Pulse_5s, PT := T#2500ms);
IF TonPulse_5s.Q THEN Pulse_5s := FALSE; END_IF;

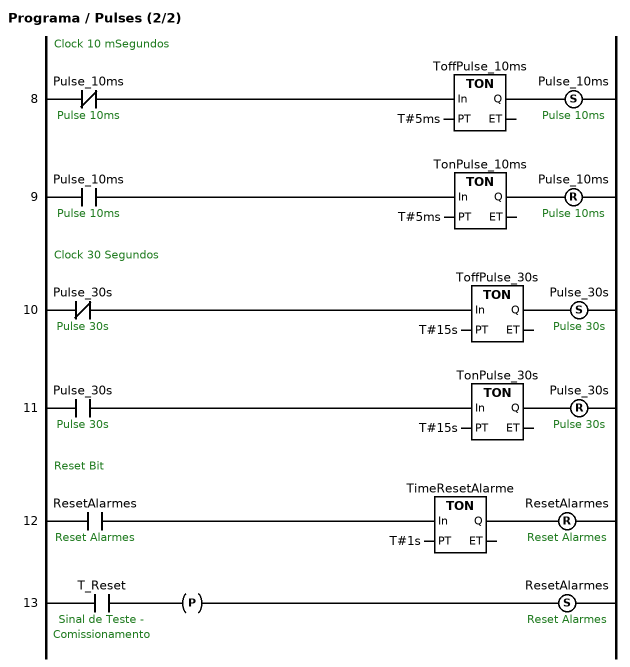
(* Rung 8: Clock 10 mSegundos *)
ToffPulse_10ms(In := NOT Pulse_10ms, PT := T#5ms);
IF ToffPulse_10ms.Q THEN Pulse_10ms := TRUE; END_IF;
(* Rung 9 *)
TonPulse_10ms(In := Pulse_10ms, PT := T#5ms);
IF TonPulse_10ms.Q THEN Pulse_10ms := FALSE; END_IF;
(* Rung 10: Clock 30 Segundos *)
ToffPulse_30s(In := NOT Pulse_30s, PT := T#15s);
IF ToffPulse_30s.Q THEN Pulse_30s := TRUE; END_IF;
(* Rung 11 *)
TonPulse_30s(In := Pulse_30s, PT := T#15s);
IF TonPulse_30s.Q THEN Pulse_30s := FALSE; END_IF;
(* Rung 12: Reset Bit *)
TimeResetAlarme(In := ResetAlarmes, PT := T#1s);
IF TimeResetAlarme.Q THEN ResetAlarmes := FALSE; END_IF;
(* Rung 13 *)
_e1(CLK := T_Reset);
IF _e1.Q THEN ResetAlarmes := TRUE; END_IF;

(* Section Geral: ladder, written here as Structured Text *)

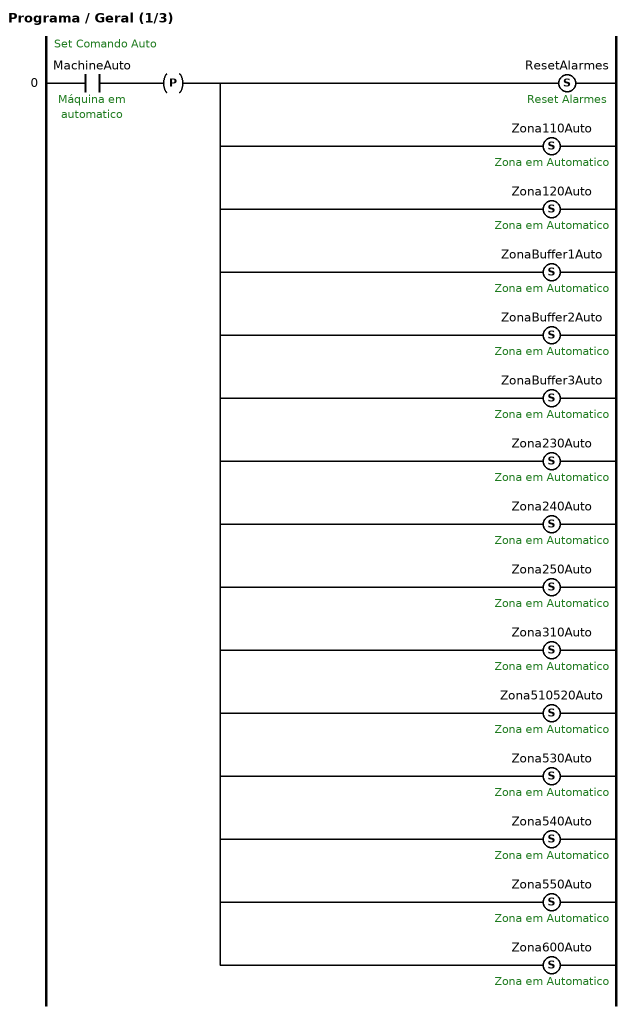
(* Rung 0: Set Comando Auto *)
_e2(CLK := MachineAuto);
IF _e2.Q THEN
    ResetAlarmes := TRUE;
    Zona110Auto := TRUE;
    Zona120Auto := TRUE;
    ZonaBuffer1Auto := TRUE;
    ZonaBuffer2Auto := TRUE;
    ZonaBuffer3Auto := TRUE;
    Zona230Auto := TRUE;
    Zona240Auto := TRUE;
    Zona250Auto := TRUE;
    Zona310Auto := TRUE;
    Zona510520Auto := TRUE;
    Zona530Auto := TRUE;
    Zona540Auto := TRUE;
    Zona550Auto := TRUE;
    Zona600Auto := TRUE;
END_IF;

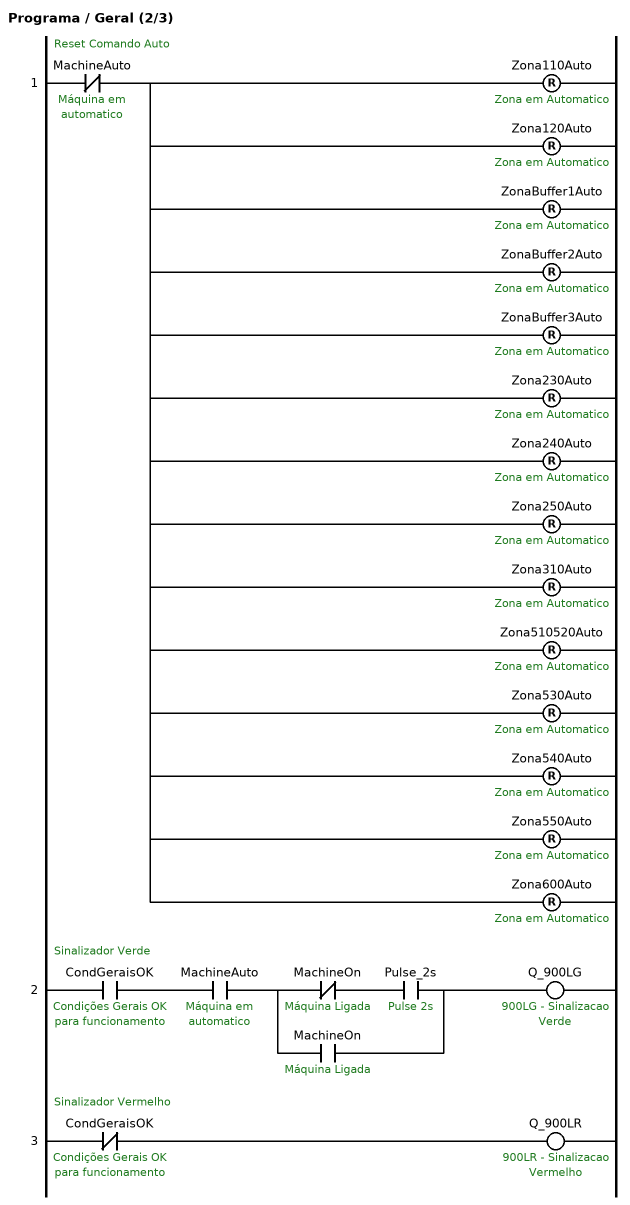
(* Rung 1: Reset Comando Auto *)
IF NOT MachineAuto THEN
    Zona110Auto := FALSE;
    Zona120Auto := FALSE;
    ZonaBuffer1Auto := FALSE;
    ZonaBuffer2Auto := FALSE;
    ZonaBuffer3Auto := FALSE;
    Zona230Auto := FALSE;
    Zona240Auto := FALSE;
    Zona250Auto := FALSE;
    Zona310Auto := FALSE;
    Zona510520Auto := FALSE;
    Zona530Auto := FALSE;
    Zona540Auto := FALSE;
    Zona550Auto := FALSE;
    Zona600Auto := FALSE;
END_IF;
(* Rung 2: Sinalizador Verde *)
Q_900LG := CondGeraisOK AND MachineAuto AND ((NOT MachineOn AND Pulse_2s) OR MachineOn);
(* Rung 3: Sinalizador Vermelho *)
Q_900LR := NOT CondGeraisOK;

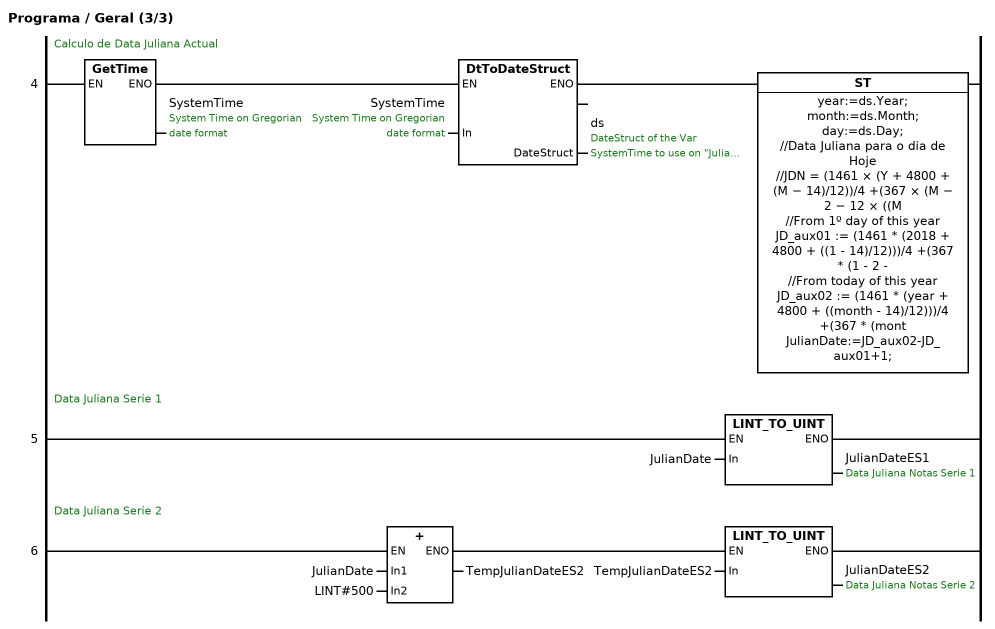
(* Rung 4: Calculo de Data Juliana Actual *)
SystemTime := GetTime();
DtToDateStruct(In := SystemTime, DateStruct => ds);
year:=ds.Year;
month:=ds.Month;
day:=ds.Day;

//Data Juliana para o dia de Hoje
//JDN = (1461 × (Y + 4800 + (M − 14)/12))/4 +(367 × (M − 2 − 12 × ((M − 14)/12)))/12 − (3 × ((Y + 4900 + (M - 14)/12)/100))/4 + D − 32075
//From 1º day of this year
JD_aux01 := (1461 * (2018 + 4800 + ((1 - 14)/12)))/4 +(367 * (1 - 2 - 12 * ((1 - 14)/12)))/12 - (3 * ((2018 + 4900 + (1 - 14)/12)/100))/4 + 1 - 32075;
//From today of this year
JD_aux02 := (1461 * (year + 4800 + ((month - 14)/12)))/4 +(367 * (month - 2 - 12 * ((month - 14)/12)))/12 - (3 * ((year + 4900 + (month - 14)/12)/100))/4 + day - 32075;

JulianDate:=JD_aux02-JD_aux01+1;
(* Rung 5: Data Juliana Serie 1 *)
JulianDateES1 := LINT_TO_UINT(In := JulianDate);
(* Rung 6: Data Juliana Serie 2 *)
TempJulianDateES2 := JulianDate + LINT#500;
JulianDateES2 := LINT_TO_UINT(In := TempJulianDateES2);

(* Section Alarmes: ladder, written here as Structured Text *)

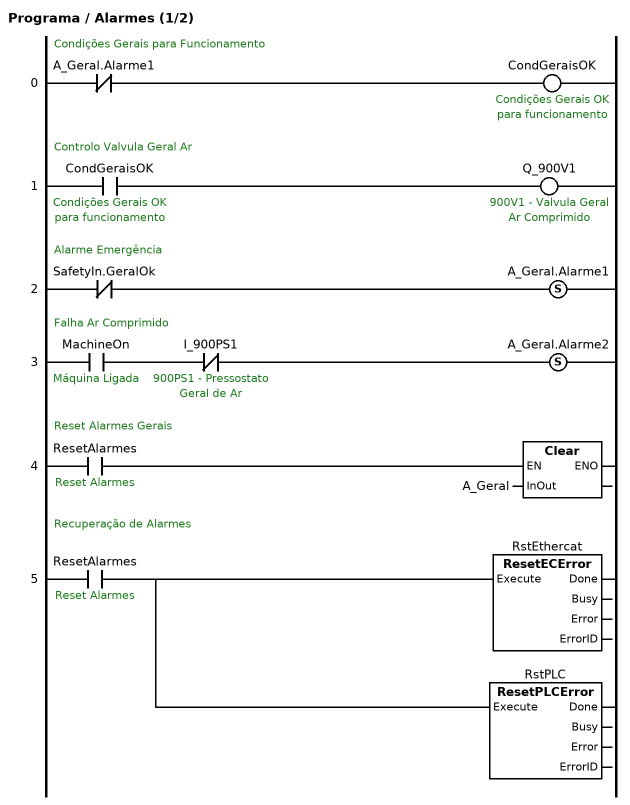
(* Rung 0: Condições Gerais para Funcionamento *)
CondGeraisOK := NOT A_Geral.Alarme1;
(* Rung 1: Controlo Valvula Geral Ar *)
Q_900V1 := CondGeraisOK;
(* Rung 2: Alarme Emergência *)
IF NOT SafetyIn.GeralOk THEN A_Geral.Alarme1 := TRUE; END_IF;
(* Rung 3: Falha Ar Comprimido *)
IF MachineOn AND NOT I_900PS1 THEN A_Geral.Alarme2 := TRUE; END_IF;
(* Rung 4: Reset Alarmes Gerais *)
IF ResetAlarmes THEN Clear(InOut := A_Geral); END_IF;
(* Rung 5: Recuperação de Alarmes *)
RstEthercat(Execute := ResetAlarmes);
RstPLC(Execute := ResetAlarmes);

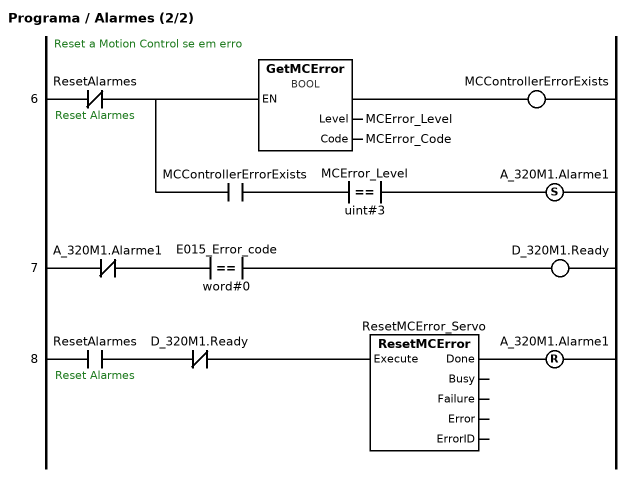
(* Rung 6: Reset a Motion Control se em erro *)
_t3 := FALSE;
IF NOT ResetAlarmes THEN _t3 := GetMCError(Level => MCError_Level, Code => MCError_Code); END_IF;
MCControllerErrorExists := _t3;
IF NOT ResetAlarmes AND MCControllerErrorExists AND (MCError_Level = uint#3) THEN
    A_320M1.Alarme1 := TRUE;
END_IF;
(* Rung 7 *)
D_320M1.Ready := NOT A_320M1.Alarme1 AND (E015_Error_code = word#0);
(* Rung 8 *)
ResetMCError_Servo(Execute := ResetAlarmes AND NOT D_320M1.Ready);
IF ResetMCError_Servo.Done THEN A_320M1.Alarme1 := FALSE; END_IF;

(* Section Ctr_110M1: ladder, written here as Structured Text *)

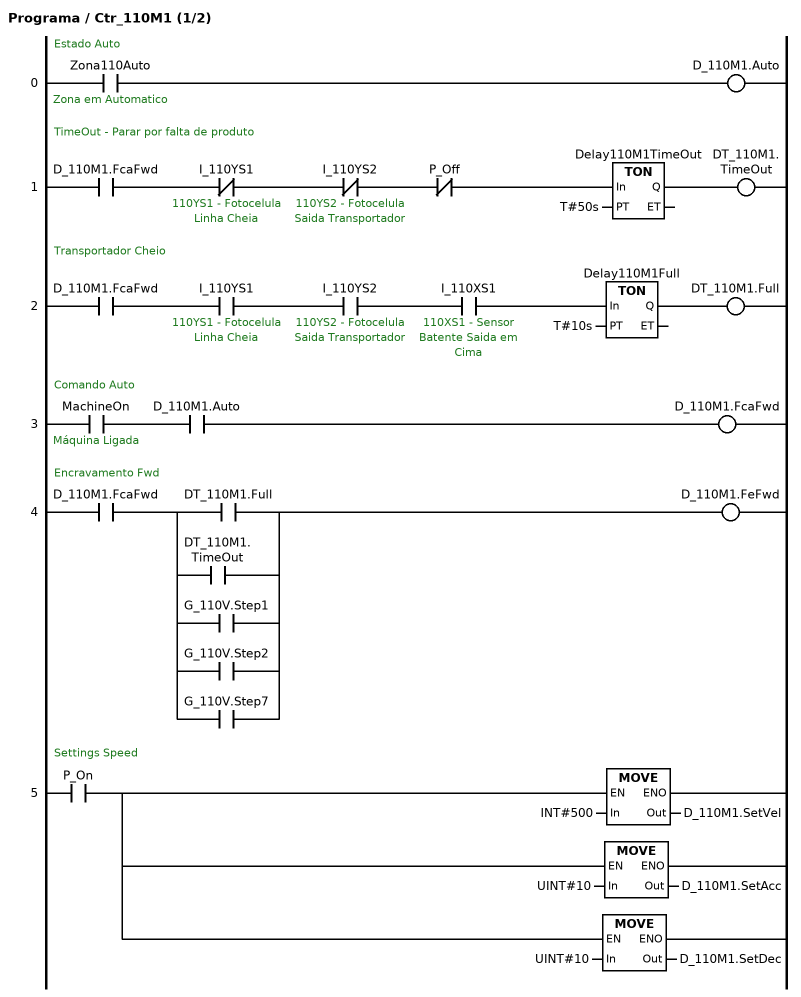
(* Rung 0: Estado Auto *)
D_110M1.Auto := Zona110Auto;
(* Rung 1: TimeOut - Parar por falta de produto *)
Delay110M1TimeOut(In := D_110M1.FcaFwd AND NOT I_110YS1 AND NOT I_110YS2 AND NOT P_Off, PT := T#50s);
DT_110M1.TimeOut := Delay110M1TimeOut.Q;
(* Rung 2: Transportador Cheio *)
Delay110M1Full(In := D_110M1.FcaFwd AND I_110YS1 AND I_110YS2 AND I_110XS1, PT := T#10s);
DT_110M1.Full := Delay110M1Full.Q;
(* Rung 3: Comando Auto *)
D_110M1.FcaFwd := MachineOn AND D_110M1.Auto;
(* Rung 4: Encravamento Fwd *)
D_110M1.FeFwd := D_110M1.FcaFwd AND (DT_110M1.Full OR DT_110M1.TimeOut OR G_110V.Step1 OR G_110V.Step2 OR G_110V.Step7);
(* Rung 5: Settings Speed *)
IF P_On THEN
    D_110M1.SetVel := INT#500;
    D_110M1.SetAcc := UINT#10;
    D_110M1.SetDec := UINT#10;
END_IF;

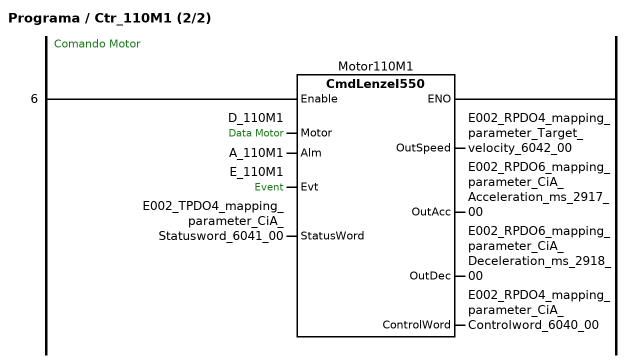
(* Rung 6: Comando Motor *)
Motor110M1(Enable := TRUE, Motor := D_110M1, Alm := A_110M1, Evt := E_110M1, StatusWord := E002_TPDO4_mapping_parameter_CiA_Statusword_6041_00, OutSpeed => E002_RPDO4_mapping_parameter_Target_velocity_6042_00, OutAcc => E002_RPDO6_mapping_parameter_CiA_Acceleration_ms_2917_00, OutDec => E002_RPDO6_mapping_parameter_CiA_Deceleration_ms_2918_00, ControlWord => E002_RPDO4_mapping_parameter_CiA_Controlword_6040_00);

(* Section Ctr_110V: ladder, written here as Structured Text *)

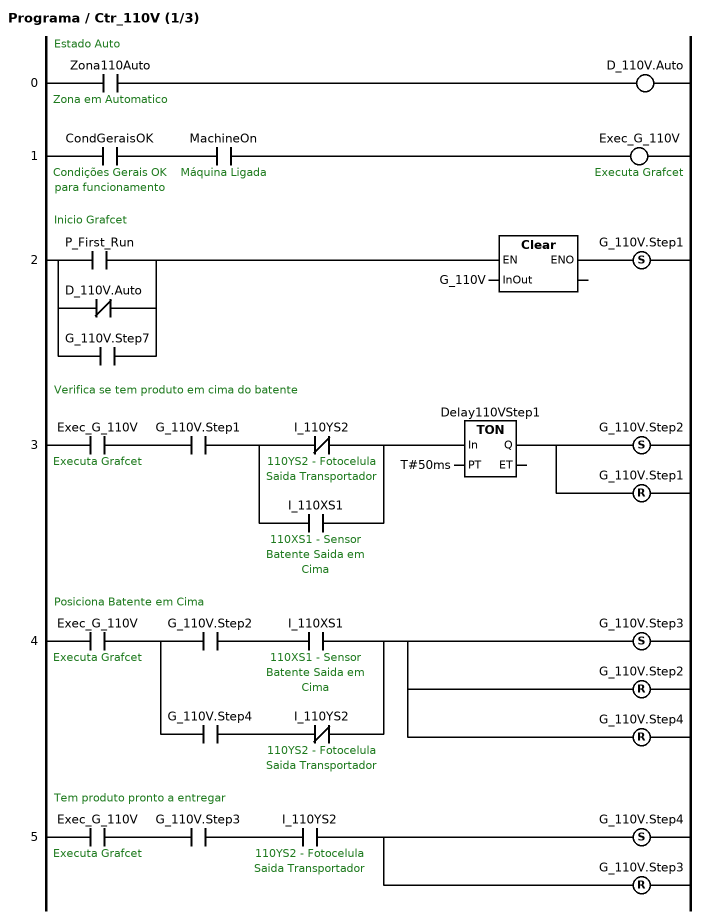
(* Rung 0: Estado Auto *)
D_110V.Auto := Zona110Auto;
(* Rung 1 *)
Exec_G_110V := CondGeraisOK AND MachineOn;
(* Rung 2: Inicio Grafcet *)
_p4 := P_First_Run OR NOT D_110V.Auto OR G_110V.Step7;
IF _p4 THEN
    Clear(InOut := G_110V);
    G_110V.Step1 := TRUE;
END_IF;
(* Rung 3: Verifica se tem produto em cima do batente *)
Delay110VStep1(In := Exec_G_110V AND G_110V.Step1 AND (NOT I_110YS2 OR I_110XS1), PT := T#50ms);
IF Delay110VStep1.Q THEN
    G_110V.Step2 := TRUE;
    G_110V.Step1 := FALSE;
END_IF;
(* Rung 4: Posiciona Batente em Cima *)
_p5 := Exec_G_110V AND ((G_110V.Step2 AND I_110XS1) OR (G_110V.Step4 AND NOT I_110YS2));
IF _p5 THEN
    G_110V.Step3 := TRUE;
    G_110V.Step2 := FALSE;
    G_110V.Step4 := FALSE;
END_IF;
(* Rung 5: Tem produto pronto a entregar *)
_p6 := Exec_G_110V AND G_110V.Step3 AND I_110YS2;
IF _p6 THEN
    G_110V.Step4 := TRUE;
    G_110V.Step3 := FALSE;
END_IF;

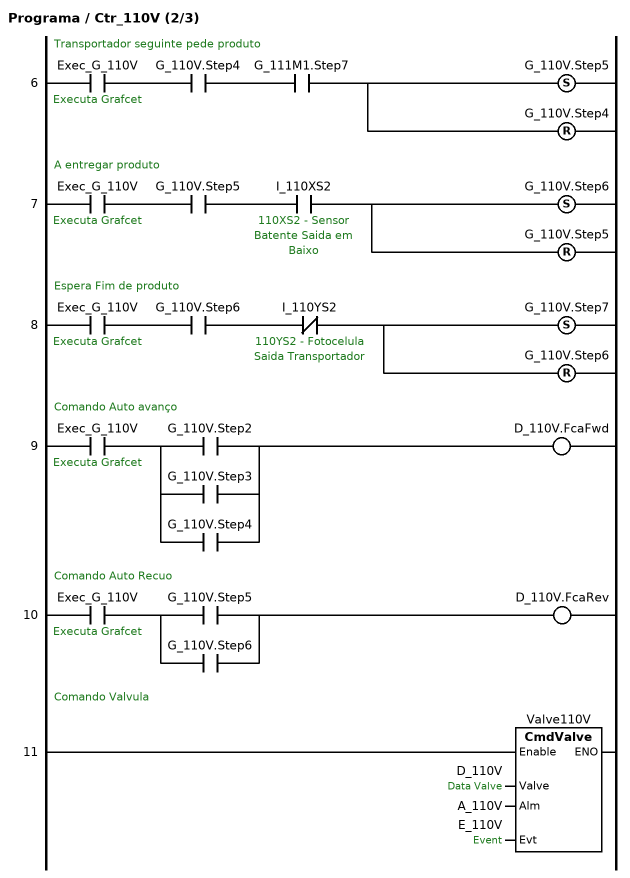
(* Rung 6: Transportador seguinte pede produto *)
_p7 := Exec_G_110V AND G_110V.Step4 AND G_111M1.Step7;
IF _p7 THEN
    G_110V.Step5 := TRUE;
    G_110V.Step4 := FALSE;
END_IF;
(* Rung 7: A entregar produto *)
_p8 := Exec_G_110V AND G_110V.Step5 AND I_110XS2;
IF _p8 THEN
    G_110V.Step6 := TRUE;
    G_110V.Step5 := FALSE;
END_IF;
(* Rung 8: Espera Fim de produto *)
_p9 := Exec_G_110V AND G_110V.Step6 AND NOT I_110YS2;
IF _p9 THEN
    G_110V.Step7 := TRUE;
    G_110V.Step6 := FALSE;
END_IF;
(* Rung 9: Comando Auto avanço *)
D_110V.FcaFwd := Exec_G_110V AND (G_110V.Step2 OR G_110V.Step3 OR G_110V.Step4);
(* Rung 10: Comando Auto Recuo *)
D_110V.FcaRev := Exec_G_110V AND (G_110V.Step5 OR G_110V.Step6);
(* Rung 11: Comando Valvula *)
Valve110V(Enable := TRUE, Valve := D_110V, Alm := A_110V, Evt := E_110V);

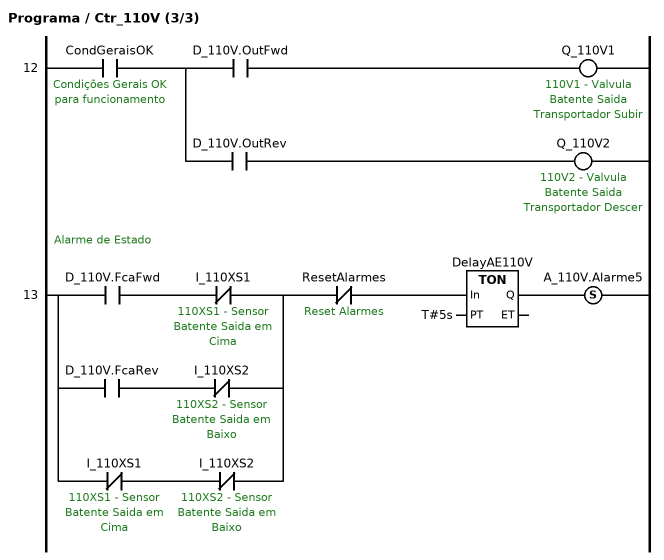
(* Rung 12 *)
Q_110V1 := CondGeraisOK AND D_110V.OutFwd;
Q_110V2 := CondGeraisOK AND D_110V.OutRev;
(* Rung 13: Alarme de Estado *)
DelayAE110V(In := ((D_110V.FcaFwd AND NOT I_110XS1) OR (D_110V.FcaRev AND NOT I_110XS2) OR (NOT I_110XS1 AND NOT I_110XS2)) AND NOT ResetAlarmes, PT := T#5s);
IF DelayAE110V.Q THEN A_110V.Alarme5 := TRUE; END_IF;

(* Section Ctr_111M1: ladder, written here as Structured Text *)

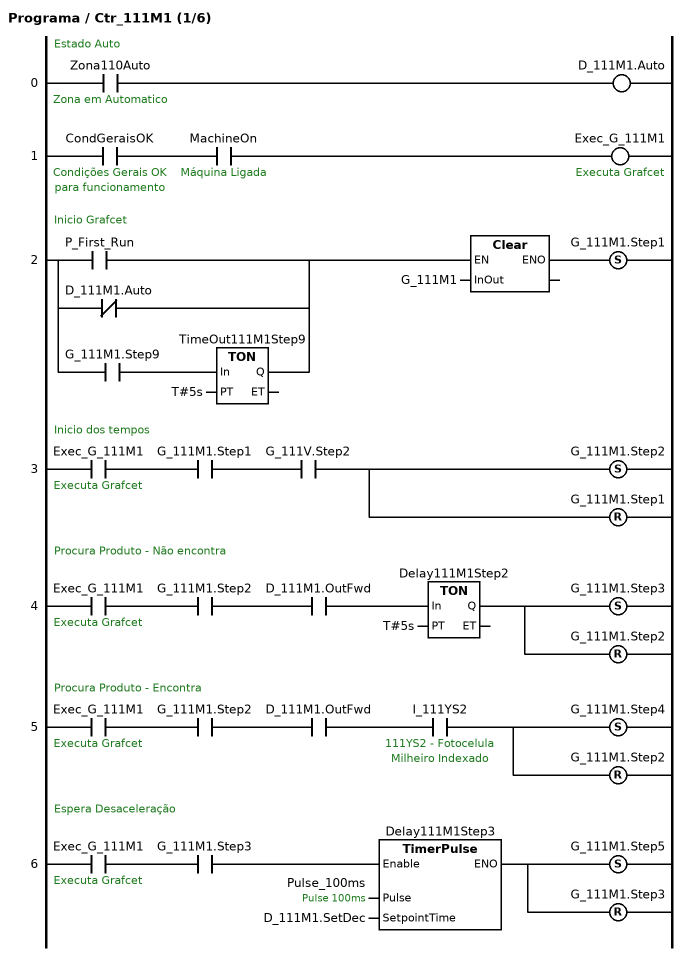
(* Rung 0: Estado Auto *)
D_111M1.Auto := Zona110Auto;
(* Rung 1 *)
Exec_G_111M1 := CondGeraisOK AND MachineOn;
(* Rung 2: Inicio Grafcet *)
TimeOut111M1Step9(In := G_111M1.Step9, PT := T#5s);
IF P_First_Run OR NOT D_111M1.Auto OR TimeOut111M1Step9.Q THEN
    Clear(InOut := G_111M1);
    G_111M1.Step1 := TRUE;
END_IF;
(* Rung 3: Inicio dos tempos *)
_p10 := Exec_G_111M1 AND G_111M1.Step1 AND G_111V.Step2;
IF _p10 THEN
    G_111M1.Step2 := TRUE;
    G_111M1.Step1 := FALSE;
END_IF;
(* Rung 4: Procura Produto - Não encontra *)
Delay111M1Step2(In := Exec_G_111M1 AND G_111M1.Step2 AND D_111M1.OutFwd, PT := T#5s);
IF Delay111M1Step2.Q THEN
    G_111M1.Step3 := TRUE;
    G_111M1.Step2 := FALSE;
END_IF;
(* Rung 5: Procura Produto - Encontra *)
_p11 := Exec_G_111M1 AND G_111M1.Step2 AND D_111M1.OutFwd AND I_111YS2;
IF _p11 THEN
    G_111M1.Step4 := TRUE;
    G_111M1.Step2 := FALSE;
END_IF;
(* Rung 6: Espera Desaceleração *)
Delay111M1Step3(Enable := Exec_G_111M1 AND G_111M1.Step3, Pulse := Pulse_100ms, SetpointTime := D_111M1.SetDec);
IF Delay111M1Step3.ENO THEN
    G_111M1.Step5 := TRUE;
    G_111M1.Step3 := FALSE;
END_IF;

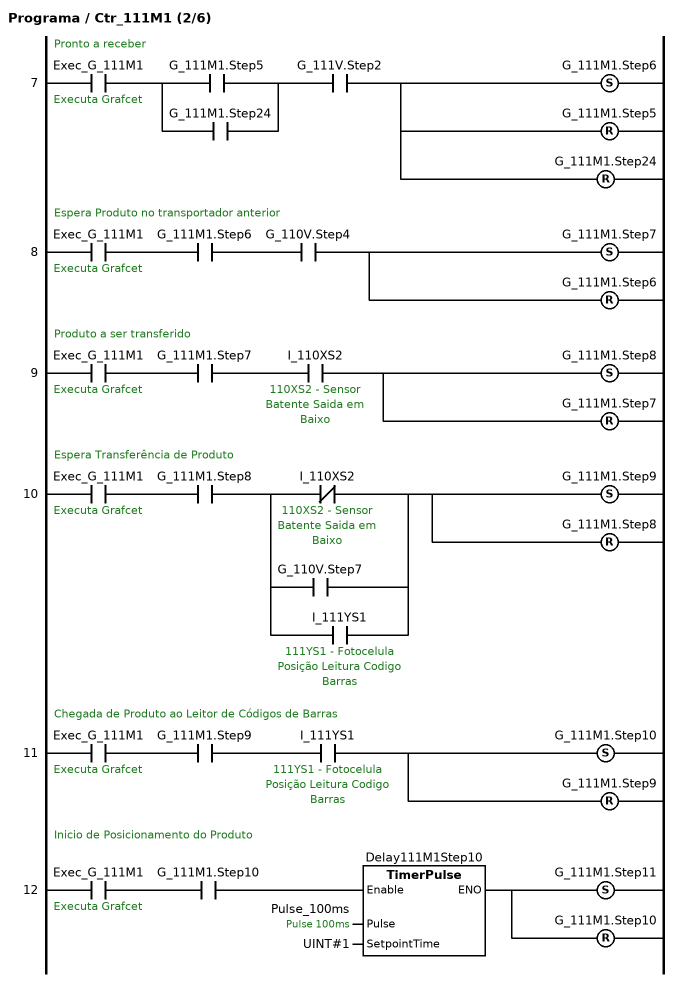
(* Rung 7: Pronto a receber *)
_p12 := Exec_G_111M1 AND (G_111M1.Step5 OR G_111M1.Step24) AND G_111V.Step2;
IF _p12 THEN
    G_111M1.Step6 := TRUE;
    G_111M1.Step5 := FALSE;
    G_111M1.Step24 := FALSE;
END_IF;
(* Rung 8: Espera Produto no transportador anterior *)
_p13 := Exec_G_111M1 AND G_111M1.Step6 AND G_110V.Step4;
IF _p13 THEN
    G_111M1.Step7 := TRUE;
    G_111M1.Step6 := FALSE;
END_IF;
(* Rung 9: Produto a ser transferido *)
_p14 := Exec_G_111M1 AND G_111M1.Step7 AND I_110XS2;
IF _p14 THEN
    G_111M1.Step8 := TRUE;
    G_111M1.Step7 := FALSE;
END_IF;
(* Rung 10: Espera Transferência de Produto *)
_p15 := Exec_G_111M1 AND G_111M1.Step8 AND (NOT I_110XS2 OR G_110V.Step7 OR I_111YS1);
IF _p15 THEN
    G_111M1.Step9 := TRUE;
    G_111M1.Step8 := FALSE;
END_IF;
(* Rung 11: Chegada de Produto ao Leitor de Códigos de Barras *)
_p16 := Exec_G_111M1 AND G_111M1.Step9 AND I_111YS1;
IF _p16 THEN
    G_111M1.Step10 := TRUE;
    G_111M1.Step9 := FALSE;
END_IF;
(* Rung 12: Inicio de Posicionamento do Produto *)
Delay111M1Step10(Enable := Exec_G_111M1 AND G_111M1.Step10, Pulse := Pulse_100ms, SetpointTime := UINT#1);
IF Delay111M1Step10.ENO THEN
    G_111M1.Step11 := TRUE;
    G_111M1.Step10 := FALSE;
END_IF;

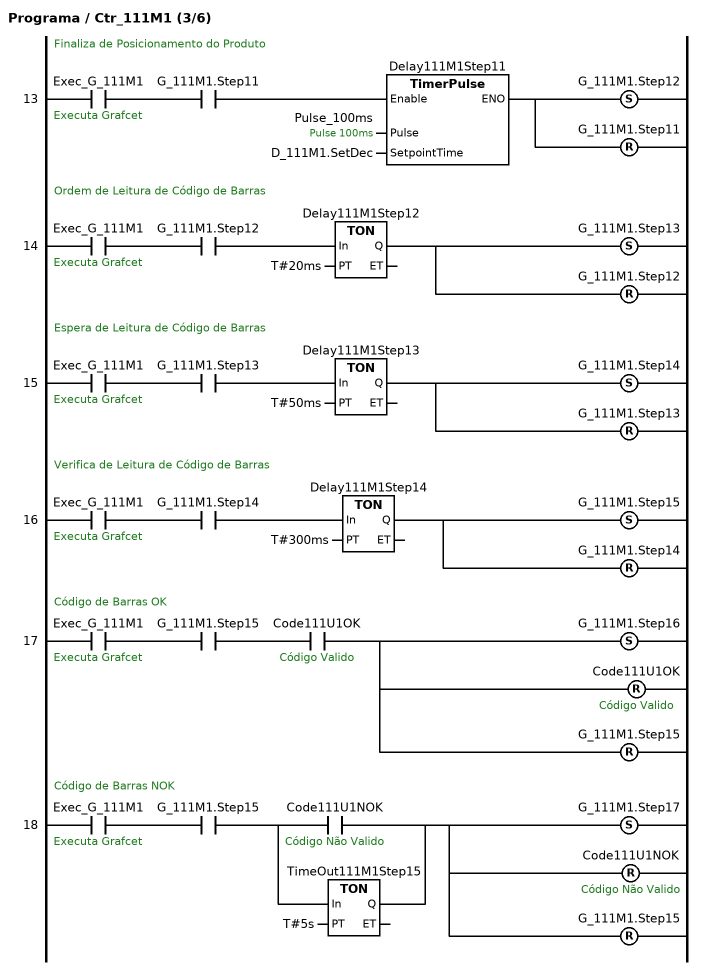
(* Rung 13: Finaliza de Posicionamento do Produto *)
Delay111M1Step11(Enable := Exec_G_111M1 AND G_111M1.Step11, Pulse := Pulse_100ms, SetpointTime := D_111M1.SetDec);
IF Delay111M1Step11.ENO THEN
    G_111M1.Step12 := TRUE;
    G_111M1.Step11 := FALSE;
END_IF;
(* Rung 14: Ordem de Leitura de Código de Barras *)
Delay111M1Step12(In := Exec_G_111M1 AND G_111M1.Step12, PT := T#20ms);
IF Delay111M1Step12.Q THEN
    G_111M1.Step13 := TRUE;
    G_111M1.Step12 := FALSE;
END_IF;
(* Rung 15: Espera de Leitura de Código de Barras *)
Delay111M1Step13(In := Exec_G_111M1 AND G_111M1.Step13, PT := T#50ms);
IF Delay111M1Step13.Q THEN
    G_111M1.Step14 := TRUE;
    G_111M1.Step13 := FALSE;
END_IF;
(* Rung 16: Verifica de Leitura de Código de Barras *)
Delay111M1Step14(In := Exec_G_111M1 AND G_111M1.Step14, PT := T#300ms);
IF Delay111M1Step14.Q THEN
    G_111M1.Step15 := TRUE;
    G_111M1.Step14 := FALSE;
END_IF;
(* Rung 17: Código de Barras OK *)
_p17 := Exec_G_111M1 AND G_111M1.Step15 AND Code111U1OK;
IF _p17 THEN
    G_111M1.Step16 := TRUE;
    Code111U1OK := FALSE;
    G_111M1.Step15 := FALSE;
END_IF;
(* Rung 18: Código de Barras NOK *)
TimeOut111M1Step15(In := Exec_G_111M1 AND G_111M1.Step15, PT := T#5s);
_p18 := (Exec_G_111M1 AND G_111M1.Step15 AND Code111U1NOK) OR TimeOut111M1Step15.Q;
IF _p18 THEN
    G_111M1.Step17 := TRUE;
    Code111U1NOK := FALSE;
    G_111M1.Step15 := FALSE;
END_IF;

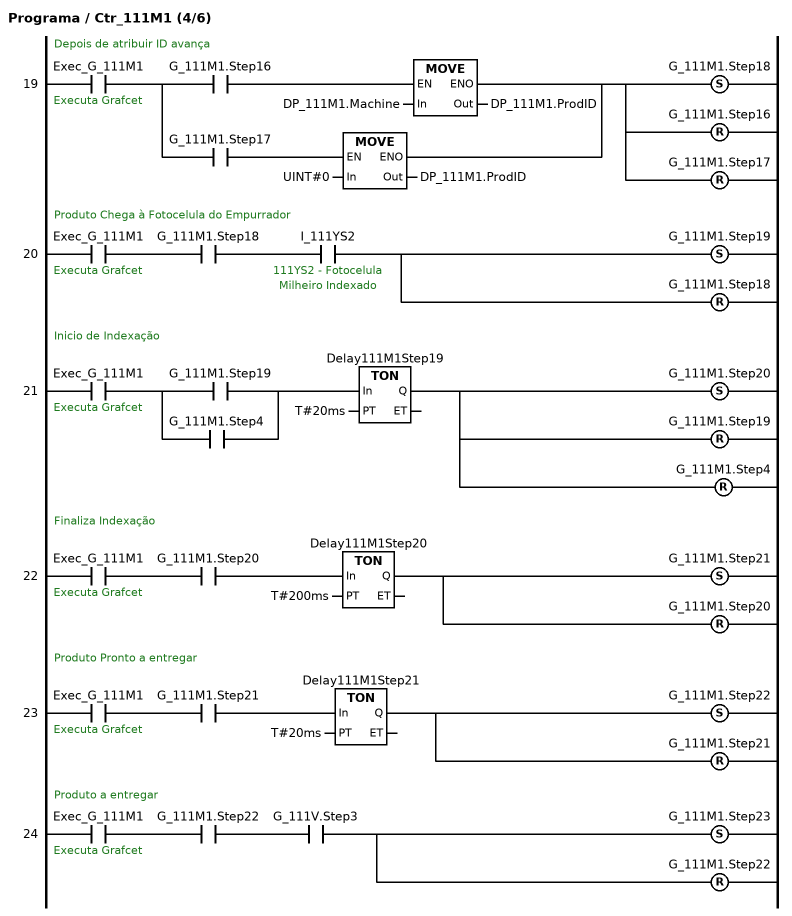
(* Rung 19: Depois de atribuir ID avança *)
IF Exec_G_111M1 AND G_111M1.Step16 THEN DP_111M1.ProdID := DP_111M1.Machine; END_IF;
IF Exec_G_111M1 AND G_111M1.Step17 THEN DP_111M1.ProdID := UINT#0; END_IF;
_p19 := Exec_G_111M1 AND (G_111M1.Step16 OR G_111M1.Step17);
IF _p19 THEN
    G_111M1.Step18 := TRUE;
    G_111M1.Step16 := FALSE;
    G_111M1.Step17 := FALSE;
END_IF;
(* Rung 20: Produto Chega à Fotocelula do Empurrador *)
_p20 := Exec_G_111M1 AND G_111M1.Step18 AND I_111YS2;
IF _p20 THEN
    G_111M1.Step19 := TRUE;
    G_111M1.Step18 := FALSE;
END_IF;
(* Rung 21: Inicio de Indexação *)
Delay111M1Step19(In := Exec_G_111M1 AND (G_111M1.Step19 OR G_111M1.Step4), PT := T#20ms);
IF Delay111M1Step19.Q THEN
    G_111M1.Step20 := TRUE;
    G_111M1.Step19 := FALSE;
    G_111M1.Step4 := FALSE;
END_IF;
(* Rung 22: Finaliza Indexação *)
Delay111M1Step20(In := Exec_G_111M1 AND G_111M1.Step20, PT := T#200ms);
IF Delay111M1Step20.Q THEN
    G_111M1.Step21 := TRUE;
    G_111M1.Step20 := FALSE;
END_IF;
(* Rung 23: Produto Pronto a entregar *)
Delay111M1Step21(In := Exec_G_111M1 AND G_111M1.Step21, PT := T#20ms);
IF Delay111M1Step21.Q THEN
    G_111M1.Step22 := TRUE;
    G_111M1.Step21 := FALSE;
END_IF;
(* Rung 24: Produto a entregar *)
_p21 := Exec_G_111M1 AND G_111M1.Step22 AND G_111V.Step3;
IF _p21 THEN
    G_111M1.Step23 := TRUE;
    G_111M1.Step22 := FALSE;
END_IF;

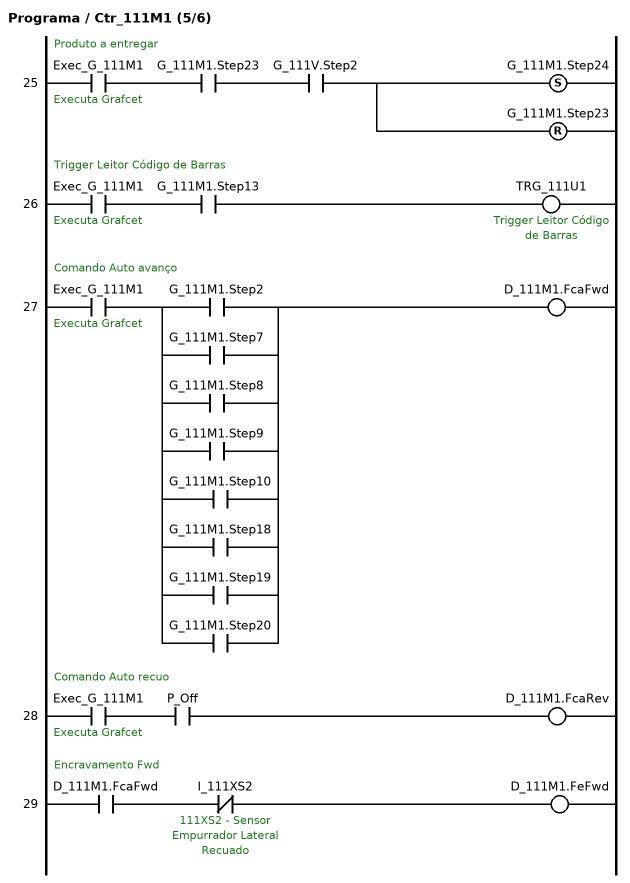
(* Rung 25: Produto a entregar *)
_p22 := Exec_G_111M1 AND G_111M1.Step23 AND G_111V.Step2;
IF _p22 THEN
    G_111M1.Step24 := TRUE;
    G_111M1.Step23 := FALSE;
END_IF;
(* Rung 26: Trigger Leitor Código de Barras *)
TRG_111U1 := Exec_G_111M1 AND G_111M1.Step13;
(* Rung 27: Comando Auto avanço *)
D_111M1.FcaFwd := Exec_G_111M1 AND (G_111M1.Step2 OR G_111M1.Step7 OR G_111M1.Step8 OR G_111M1.Step9 OR G_111M1.Step10 OR G_111M1.Step18 OR G_111M1.Step19 OR G_111M1.Step20);
(* Rung 28: Comando Auto recuo *)
D_111M1.FcaRev := Exec_G_111M1 AND P_Off;
(* Rung 29: Encravamento Fwd *)
D_111M1.FeFwd := D_111M1.FcaFwd AND NOT I_111XS2;

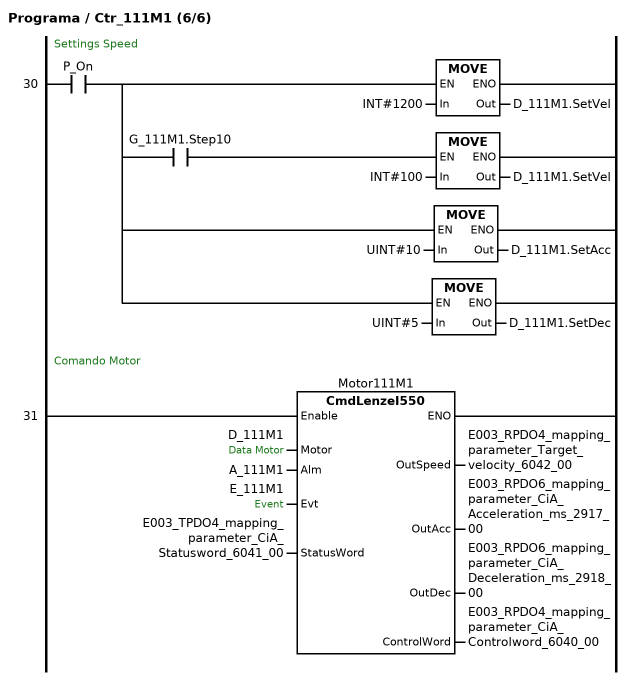
(* Rung 30: Settings Speed *)
IF P_On THEN D_111M1.SetVel := INT#1200; END_IF;
IF P_On AND G_111M1.Step10 THEN D_111M1.SetVel := INT#100; END_IF;
IF P_On THEN
    D_111M1.SetAcc := UINT#10;
    D_111M1.SetDec := UINT#5;
END_IF;
(* Rung 31: Comando Motor *)
Motor111M1(Enable := TRUE, Motor := D_111M1, Alm := A_111M1, Evt := E_111M1, StatusWord := E003_TPDO4_mapping_parameter_CiA_Statusword_6041_00, OutSpeed => E003_RPDO4_mapping_parameter_Target_velocity_6042_00, OutAcc => E003_RPDO6_mapping_parameter_CiA_Acceleration_ms_2917_00, OutDec => E003_RPDO6_mapping_parameter_CiA_Deceleration_ms_2918_00, ControlWord => E003_RPDO4_mapping_parameter_CiA_Controlword_6040_00);

(* Section Data_111U1: ladder, written here as Structured Text *)

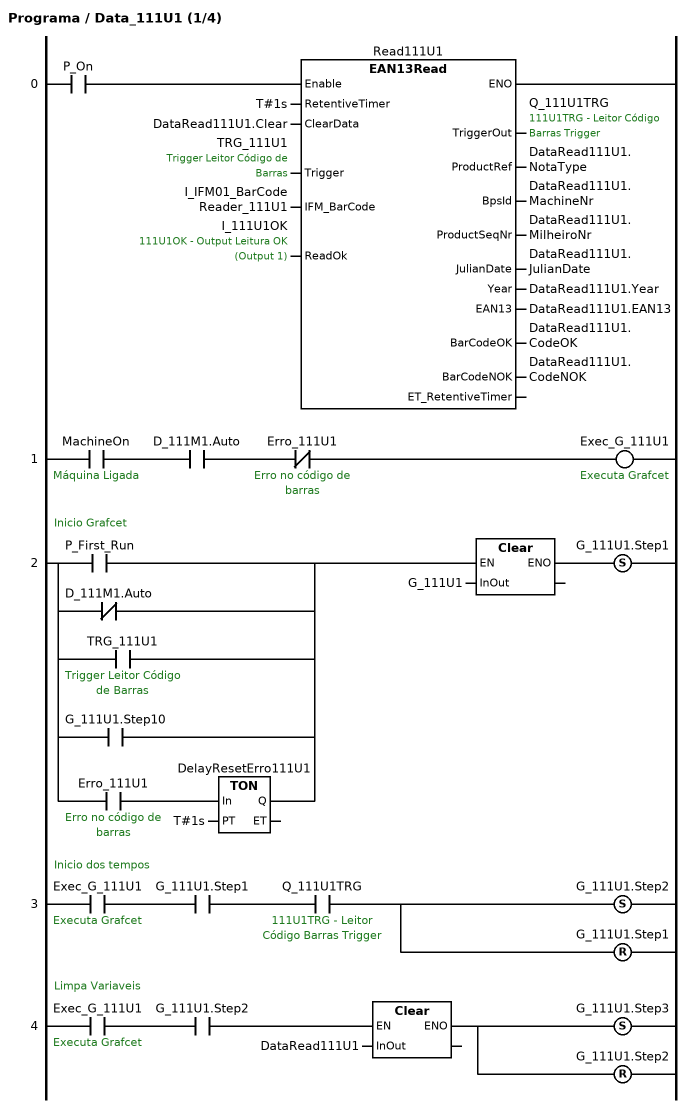
(* Rung 0 *)
Read111U1(Enable := P_On, RetentiveTimer := T#1s, ClearData := DataRead111U1.Clear, Trigger := TRG_111U1, IFM_BarCode := I_IFM01_BarCodeReader_111U1, ReadOk := I_111U1OK, TriggerOut => Q_111U1TRG, ProductRef => DataRead111U1.NotaType, BpsId => DataRead111U1.MachineNr, ProductSeqNr => DataRead111U1.MilheiroNr, JulianDate => DataRead111U1.JulianDate, Year => DataRead111U1.Year, EAN13 => DataRead111U1.EAN13, BarCodeOK => DataRead111U1.CodeOK, BarCodeNOK => DataRead111U1.CodeNOK);
(* Rung 1 *)
Exec_G_111U1 := MachineOn AND D_111M1.Auto AND NOT Erro_111U1;
(* Rung 2: Inicio Grafcet *)
DelayResetErro111U1(In := Erro_111U1, PT := T#1s);
_p23 := P_First_Run OR NOT D_111M1.Auto OR TRG_111U1 OR G_111U1.Step10 OR DelayResetErro111U1.Q;
IF _p23 THEN
    Clear(InOut := G_111U1);
    G_111U1.Step1 := TRUE;
END_IF;
(* Rung 3: Inicio dos tempos *)
_p24 := Exec_G_111U1 AND G_111U1.Step1 AND Q_111U1TRG;
IF _p24 THEN
    G_111U1.Step2 := TRUE;
    G_111U1.Step1 := FALSE;
END_IF;
(* Rung 4: Limpa Variaveis *)
IF Exec_G_111U1 AND G_111U1.Step2 THEN Clear(InOut := DataRead111U1); END_IF;
_p25 := Exec_G_111U1 AND G_111U1.Step2;
IF _p25 THEN
    G_111U1.Step3 := TRUE;
    G_111U1.Step2 := FALSE;
END_IF;

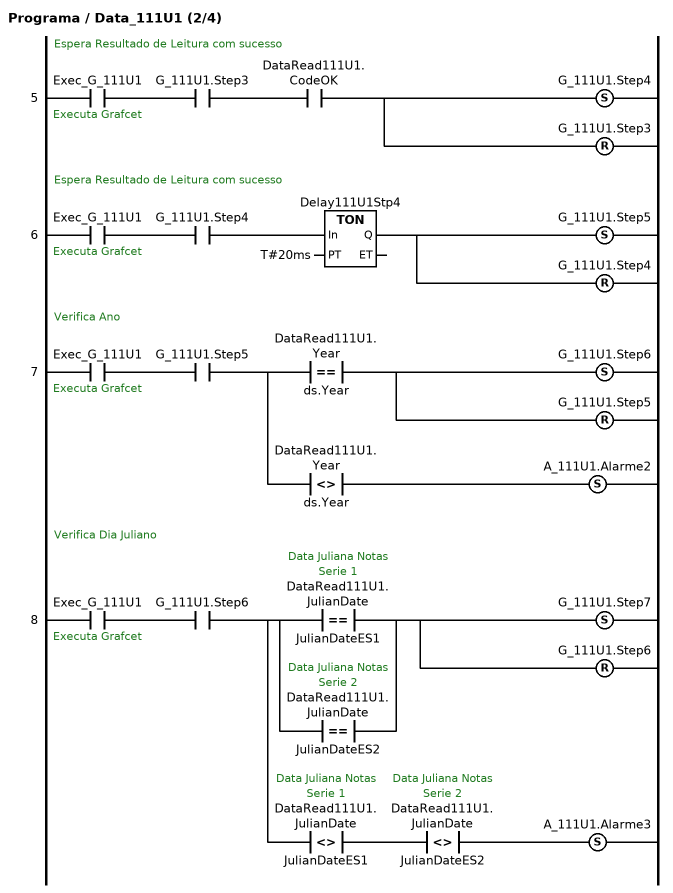
(* Rung 5: Espera Resultado de Leitura com sucesso *)
_p26 := Exec_G_111U1 AND G_111U1.Step3 AND DataRead111U1.CodeOK;
IF _p26 THEN
    G_111U1.Step4 := TRUE;
    G_111U1.Step3 := FALSE;
END_IF;
(* Rung 6: Espera Resultado de Leitura com sucesso *)
Delay111U1Stp4(In := Exec_G_111U1 AND G_111U1.Step4, PT := T#20ms);
IF Delay111U1Stp4.Q THEN
    G_111U1.Step5 := TRUE;
    G_111U1.Step4 := FALSE;
END_IF;
(* Rung 7: Verifica Ano *)
_p27 := Exec_G_111U1 AND G_111U1.Step5 AND (DataRead111U1.Year = ds.Year);
_p28 := Exec_G_111U1 AND G_111U1.Step5;
IF _p27 THEN
    G_111U1.Step6 := TRUE;
    G_111U1.Step5 := FALSE;
END_IF;
IF _p28 AND (DataRead111U1.Year <> ds.Year) THEN A_111U1.Alarme2 := TRUE; END_IF;
(* Rung 8: Verifica Dia Juliano *)
_p29 := Exec_G_111U1 AND G_111U1.Step6 AND ((DataRead111U1.JulianDate = JulianDateES1) OR (DataRead111U1.JulianDate = JulianDateES2));
_p30 := Exec_G_111U1 AND G_111U1.Step6;
IF _p29 THEN
    G_111U1.Step7 := TRUE;
    G_111U1.Step6 := FALSE;
END_IF;
IF _p30 AND (DataRead111U1.JulianDate <> JulianDateES1) AND (DataRead111U1.JulianDate <> JulianDateES2) THEN
    A_111U1.Alarme3 := TRUE;
END_IF;

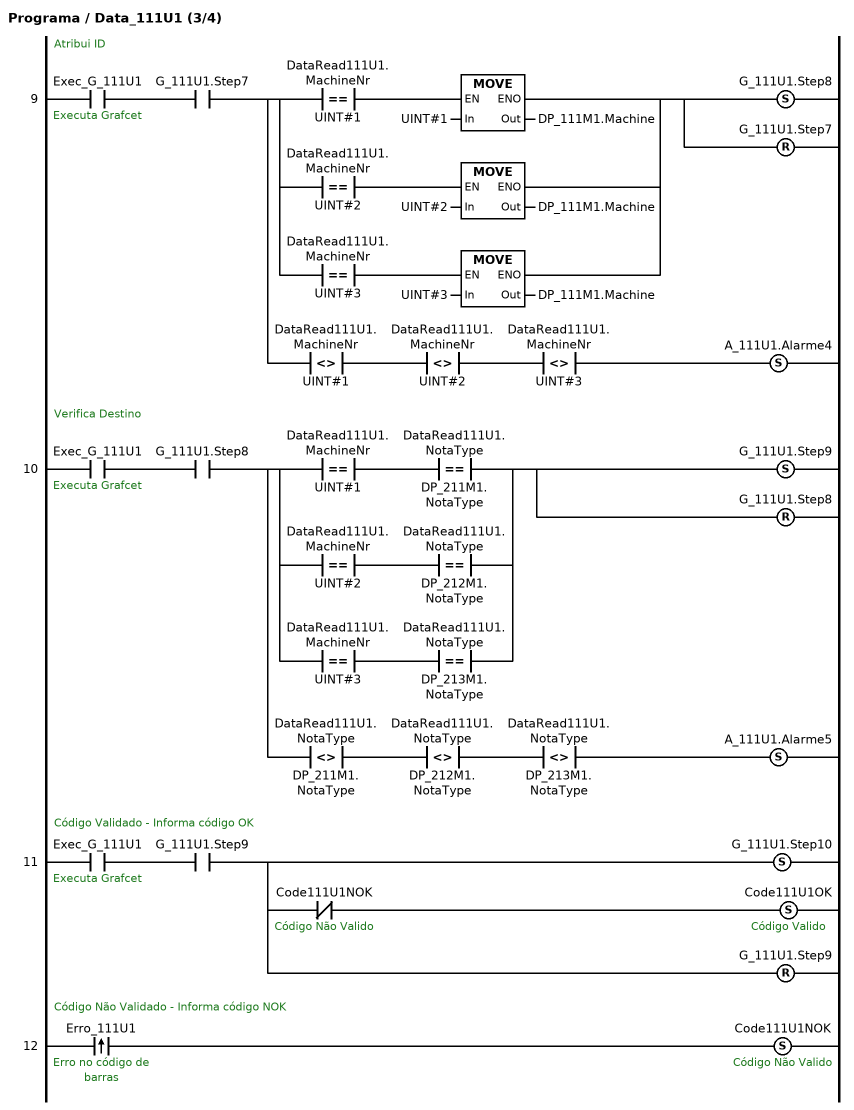
(* Rung 9: Atribui ID *)
IF Exec_G_111U1 AND G_111U1.Step7 AND (DataRead111U1.MachineNr = UINT#1) THEN
    DP_111M1.Machine := UINT#1;
END_IF;
IF Exec_G_111U1 AND G_111U1.Step7 AND (DataRead111U1.MachineNr = UINT#2) THEN
    DP_111M1.Machine := UINT#2;
END_IF;
IF Exec_G_111U1 AND G_111U1.Step7 AND (DataRead111U1.MachineNr = UINT#3) THEN
    DP_111M1.Machine := UINT#3;
END_IF;
_p31 := Exec_G_111U1 AND G_111U1.Step7 AND ((DataRead111U1.MachineNr = UINT#1) OR (DataRead111U1.MachineNr = UINT#2) OR (DataRead111U1.MachineNr = UINT#3));
_p32 := Exec_G_111U1 AND G_111U1.Step7;
IF _p31 THEN
    G_111U1.Step8 := TRUE;
    G_111U1.Step7 := FALSE;
END_IF;
IF _p32 AND (DataRead111U1.MachineNr <> UINT#1) AND (DataRead111U1.MachineNr <> UINT#2) AND (DataRead111U1.MachineNr <> UINT#3) THEN
    A_111U1.Alarme4 := TRUE;
END_IF;
(* Rung 10: Verifica Destino *)
_p33 := Exec_G_111U1 AND G_111U1.Step8 AND (((DataRead111U1.MachineNr = UINT#1) AND (DataRead111U1.NotaType = DP_211M1.NotaType)) OR ((DataRead111U1.MachineNr = UINT#2) AND (DataRead111U1.NotaType = DP_212M1.NotaType)) OR ((DataRead111U1.MachineNr = UINT#3) AND (DataRead111U1.NotaType = DP_213M1.NotaType)));
_p34 := Exec_G_111U1 AND G_111U1.Step8;
IF _p33 THEN
    G_111U1.Step9 := TRUE;
    G_111U1.Step8 := FALSE;
END_IF;
IF _p34 AND (DataRead111U1.NotaType <> DP_211M1.NotaType) AND (DataRead111U1.NotaType <> DP_212M1.NotaType) AND (DataRead111U1.NotaType <> DP_213M1.NotaType) THEN
    A_111U1.Alarme5 := TRUE;
END_IF;
(* Rung 11: Código Validado - Informa código OK *)
_p35 := Exec_G_111U1 AND G_111U1.Step9;
IF _p35 THEN G_111U1.Step10 := TRUE; END_IF;
IF _p35 AND NOT Code111U1NOK THEN Code111U1OK := TRUE; END_IF;
IF _p35 THEN G_111U1.Step9 := FALSE; END_IF;
(* Rung 12: Código Não Validado - Informa código NOK *)
_e36(CLK := Erro_111U1);
IF _e36.Q THEN Code111U1NOK := TRUE; END_IF;

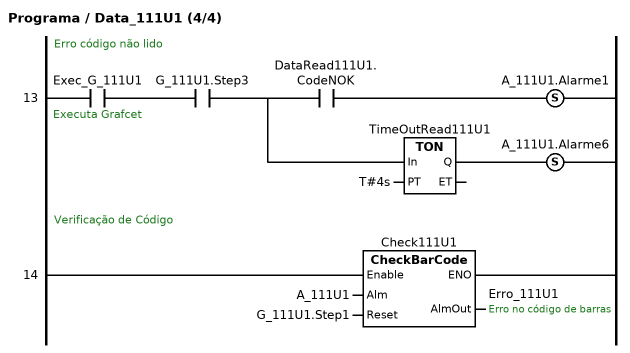
(* Rung 13: Erro código não lido *)
IF Exec_G_111U1 AND G_111U1.Step3 AND DataRead111U1.CodeNOK THEN A_111U1.Alarme1 := TRUE; END_IF;
TimeOutRead111U1(In := Exec_G_111U1 AND G_111U1.Step3, PT := T#4s);
IF TimeOutRead111U1.Q THEN A_111U1.Alarme6 := TRUE; END_IF;
(* Rung 14: Verificação de Código *)
Check111U1(Enable := TRUE, Alm := A_111U1, Reset := G_111U1.Step1, AlmOut => Erro_111U1);

(* Section Ctr_111V: ladder, written here as Structured Text *)

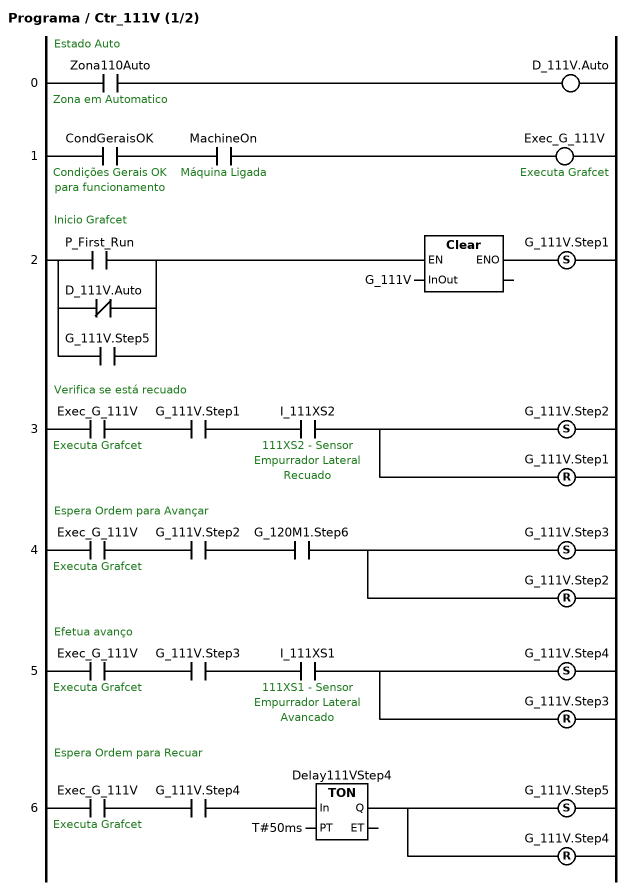
(* Rung 0: Estado Auto *)
D_111V.Auto := Zona110Auto;
(* Rung 1 *)
Exec_G_111V := CondGeraisOK AND MachineOn;
(* Rung 2: Inicio Grafcet *)
_p37 := P_First_Run OR NOT D_111V.Auto OR G_111V.Step5;
IF _p37 THEN
    Clear(InOut := G_111V);
    G_111V.Step1 := TRUE;
END_IF;
(* Rung 3: Verifica se está recuado *)
_p38 := Exec_G_111V AND G_111V.Step1 AND I_111XS2;
IF _p38 THEN
    G_111V.Step2 := TRUE;
    G_111V.Step1 := FALSE;
END_IF;
(* Rung 4: Espera Ordem para Avançar *)
_p39 := Exec_G_111V AND G_111V.Step2 AND G_120M1.Step6;
IF _p39 THEN
    G_111V.Step3 := TRUE;
    G_111V.Step2 := FALSE;
END_IF;
(* Rung 5: Efetua avanço *)
_p40 := Exec_G_111V AND G_111V.Step3 AND I_111XS1;
IF _p40 THEN
    G_111V.Step4 := TRUE;
    G_111V.Step3 := FALSE;
END_IF;
(* Rung 6: Espera Ordem para Recuar *)
Delay111VStep4(In := Exec_G_111V AND G_111V.Step4, PT := T#50ms);
IF Delay111VStep4.Q THEN
    G_111V.Step5 := TRUE;
    G_111V.Step4 := FALSE;
END_IF;

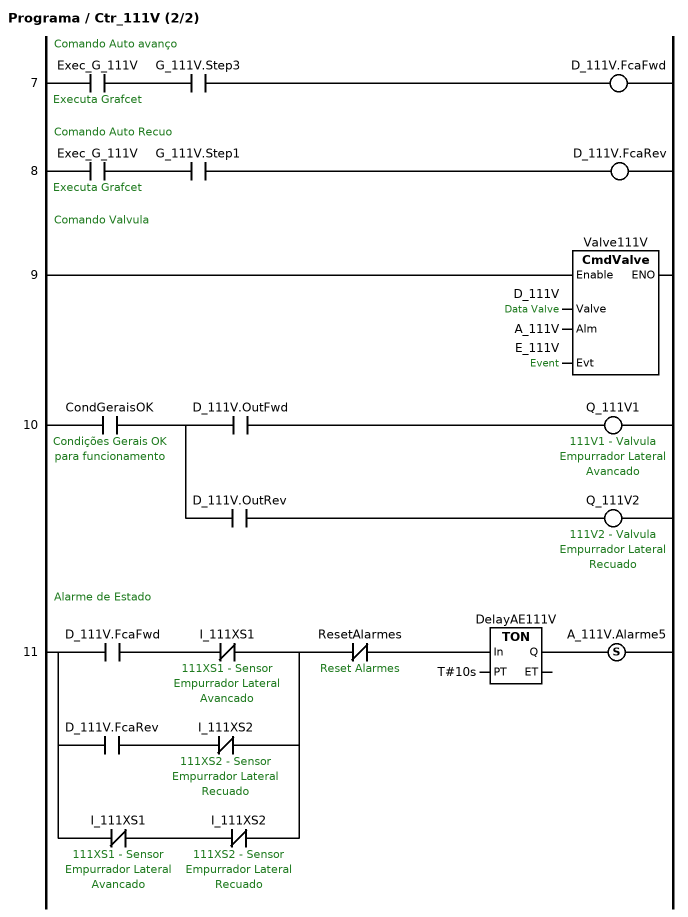
(* Rung 7: Comando Auto avanço *)
D_111V.FcaFwd := Exec_G_111V AND G_111V.Step3;
(* Rung 8: Comando Auto Recuo *)
D_111V.FcaRev := Exec_G_111V AND G_111V.Step1;
(* Rung 9: Comando Valvula *)
Valve111V(Enable := TRUE, Valve := D_111V, Alm := A_111V, Evt := E_111V);
(* Rung 10 *)
Q_111V1 := CondGeraisOK AND D_111V.OutFwd;
Q_111V2 := CondGeraisOK AND D_111V.OutRev;
(* Rung 11: Alarme de Estado *)
DelayAE111V(In := ((D_111V.FcaFwd AND NOT I_111XS1) OR (D_111V.FcaRev AND NOT I_111XS2) OR (NOT I_111XS1 AND NOT I_111XS2)) AND NOT ResetAlarmes, PT := T#10s);
IF DelayAE111V.Q THEN A_111V.Alarme5 := TRUE; END_IF;

(* Section Ctr_120M1: ladder, written here as Structured Text *)

